LIN {X 0,Y 418.219,Z 282.716,A -85,B 0,C 180,E1 -10133.218,E2 -10133.218} C_VEL
LIN {X 0,Y 423.907,Z 299.688,A -85,B 0,C 180,E1 -10135.991,E2 -10135.991} C_VEL
LIN {X 0,Y 426.524,Z 308.051,A -85,B 0,C 180,E1 -10137.245,E2 -10137.245} C_VEL
LIN {X 0,Y 433.499,Z 322.682,A -85,B 0,C 180,E1 -10138.112,E2 -10138.112} C_VEL
LIN {X 0,Y 436.744,Z 342.587,A -85,B 0,C 180,E1 -10138.75,E2 -10138.75} C_VEL
LIN {X 0,Y 433.204,Z 515.05,A -85,B 0,C 180,E1 -10141.722,E2 -10141.722} C_VEL
LIN {X 0,Y 432.227,Z 531.382,A -85,B 0,C 180,E1 -10142.163,E2 -10142.163} C_VEL
LIN {X 0,Y 431.166,Z 547.235,A -85,B 0,C 180,E1 -10142.78,E2 -10142.78} C_VEL
LIN {X 0,Y 429.887,Z 562.43,A -85,B 0,C 180,E1 -10143.545,E2 -10143.545} C_VEL
LIN {X 0,Y 428.397,Z 577.584,A -85,B 0,C 180,E1 -10144.505,E2 -10144.505} C_VEL
LIN {X 0,Y 426.712,Z 592.691,A -85,B 0,C 180,E1 -10145.685,E2 -10145.685} C_VEL
LIN {X 0,Y 425.026,Z 606.696,A -85,B 0,C 180,E1 -10147.005,E2 -10147.005} C_VEL
LIN {X 0,Y 423.355,Z 620.63,A -85,B 0,C 180,E1 -10148.579,E2 -10148.579} C_VEL
LIN {X 0,Y 422.008,Z 631.644,A -85,B 0,C 180,E1 -10150.038,E2 -10150.038} C_VEL
LIN {X 0,Y 420.616,Z 642.771,A -85,B 0,C 180,E1 -10151.768,E2 -10151.768} C_VEL
LIN {X 0,Y 419.527,Z 653.245,A -85,B 0,C 180,E1 -10153.704,E2 -10153.704} C_VEL
LIN {X 0,Y 418.528,Z 662.163,A -85,B 0,C 180,E1 -10155.66,E2 -10155.66} C_VEL
LIN {X 0,Y 418.017,Z 668.813,A -85,B 0,C 180,E1 -10157.375,E2 -10157.375} C_VEL
LIN {X 0,Y 417.396,Z 676.506,A -85,B 0,C 180,E1 -10159.817,E2 -10159.817} C_VEL
LIN {X 0,Y 417.147,Z 682.365,A -85,B 0,C 180,E1 -10162.254,E2 -10162.254} C_VEL
LIN {X 0,Y 417.065,Z 685.793,A -85,B 0,C 180,E1 -10164.197,E2 -10164.197} C_VEL
LIN {X 0,Y 416.984,Z 688.283,A -85,B 0,C 180,E1 -10166.134,E2 -10166.134} C_VEL
LIN {X 0,Y 417.046,Z 689.691,A -85,B 0,C 180,E1 -10168.069,E2 -10168.069} C_VEL
LIN {X 0,Y 416.999,Z 690.219,A -85,B 0,C 180,E1 -10170,E2 -10170} C_VEL
LIN {X 0,Y 417.046,Z 689.689,A -85,B 0,C 180,E1 -10171.931,E2 -10171.931} C_VEL
LIN {X 0,Y 416.984,Z 688.278,A -85,B 0,C 180,E1 -10173.866,E2 -10173.866} C_VEL
LIN {X 0,Y 417.138,Z 685.094,A -85,B 0,C 180,E1 -10176.261,E2 -10176.261} C_VEL
LIN {X 0,Y 417.2,Z 681.284,A -85,B 0,C 180,E1 -10178.232,E2 -10178.232} C_VEL
LIN {X 0,Y 417.396,Z 676.5,A -85,B 0,C 180,E1 -10180.183,E2 -10180.183} C_VEL
LIN {X 0,Y 418.01,Z 668.8,A -85,B 0,C 180,E1 -10182.625,E2 -10182.625} C_VEL
LIN {X 0,Y 418.753,Z 660.111,A -85,B 0,C 180,E1 -10184.829,E2 -10184.829} C_VEL
LIN {X 0,Y 419.759,Z 650.785,A -85,B 0,C 180,E1 -10186.778,E2 -10186.778} C_VEL
LIN {X 0,Y 420.799,Z 641.099,A -85,B 0,C 180,E1 -10188.501,E2 -10188.501} C_VEL
LIN {X 0,Y 422.21,Z 629.874,A -85,B 0,C 180,E1 -10190.206,E2 -10190.206} C_VEL
LIN {X 0,Y 423.641,Z 618.18,A -85,B 0,C 180,E1 -10191.719,E2 -10191.719} C_VEL
LIN {X 0,Y 425.161,Z 605.467,A -85,B 0,C 180,E1 -10193.116,E2 -10193.116} C_VEL
LIN {X 0,Y 426.836,Z 591.192,A -85,B 0,C 180,E1 -10194.437,E2 -10194.437} C_VEL
LIN {X 0,Y 428.496,Z 576.432,A -85,B 0,C 180,E1 -10195.567,E2 -10195.567} C_VEL
LIN {X 0,Y 429.977,Z 561.328,A -85,B 0,C 180,E1 -10196.514,E2 -10196.514} C_VEL
LIN {X 0,Y 431.288,Z 545.808,A -85,B 0,C 180,E1 -10197.278,E2 -10197.278} C_VEL
LIN {X 0,Y 432.34,Z 530.29,A -85,B 0,C 180,E1 -10197.862,E2 -10197.862} C_VEL
LIN {X 0,Y 433.159,Z 515.027,A -85,B 0,C 180,E1 -10198.276,E2 -10198.276} C_VEL
LIN {X 0,Y 436.324,Z 361.208,A -85,B 0,C 180,E1 -10200.926,E2 -10200.926} C_VEL
LIN {X 0,Y 436.722,Z 342.306,A -85,B 0,C 180,E1 -10201.25,E2 -10201.25} C_VEL
LIN {X 0,Y 433.182,Z 322.055,A -85,B 0,C 180,E1 -10201.918,E2 -10201.918} C_VEL
LIN {X 0,Y 426.335,Z 307.543,A -85,B 0,C 180,E1 -10202.784,E2 -10202.784} C_VEL
LIN {X 0,Y 421.419,Z 292.204,A -85,B 0,C 180,E1 -10205.198,E2 -10205.198} C_VEL
LIN {X 0,Y 418.229,Z 282.702,A -85,B 0,C 180,E1 -10206.779,E2 -10206.779} C_VEL
LIN {X 0,Y 418.252,Z 282.699,A -85,B 0,C 180,E1 -10209.681,E2 -10209.681} C_VEL
LIN {X 0,Y 418.23,Z 282.699,A -85,B 0,C 180,E1 -10212.322,E2 -10212.322} C_VEL
LIN {X 0,Y 418.236,Z 282.699,A -85,B 0,C 180,E1 -10215.109,E2 -10215.109} C_VEL
LIN {X 0,Y 418.237,Z 282.694,A -85,B 0,C 180,E1 -10217.767,E2 -10217.767} C_VEL
LIN {X 0,Y 418.246,Z 282.692,A -85,B 0,C 180,E1 -10220.62,E2 -10220.62} C_VEL
LIN {X 0,Y 418.241,Z 282.695,A -85,B 0,C 180,E1 -10223.976,E2 -10223.976} C_VEL
LIN {X 0,Y 418.255,Z 282.695,A -85,B 0,C 180,E1 -10227.156,E2 -10227.156} C_VEL
LIN {X 0,Y 418.266,Z 282.695,A -85,B 0,C 180,E1 -10230.895,E2 -10230.895} C_VEL
LIN {X 0,Y 418.268,Z 282.694,A -85,B 0,C 180,E1 -10234.096,E2 -10234.096} C_VEL
LIN {X 0,Y 418.236,Z 282.701,A -85,B 0,C 180,E1 -10237.264,E2 -10237.264} C_VEL
LIN {X 0,Y 418.28,Z 282.673,A -85,B 0,C 180,E1 -10240.364,E2 -10240.364} C_VEL
LIN {X 0,Y 418.314,Z 282.69,A -85,B 0,C 180,E1 -10243.405,E2 -10243.405} C_VEL
LIN {X 0,Y 418.344,Z 282.666,A -85,B 0,C 180,E1 -10246.999,E2 -10246.999} C_VEL
LIN {X 0,Y 418.339,Z 282.685,A -85,B 0,C 180,E1 -10250.329,E2 -10250.329} C_VEL
LIN {X 0,Y 418.491,Z 282.646,A -85,B 0,C 180,E1 -10253.249,E2 -10253.249} C_VEL
LIN {X 0,Y 418.338,Z 282.676,A -85,B 0,C 180,E1 -10255.182,E2 -10255.182} C_VEL
LIN {X 0,Y 418.542,Z 282.658,A -85,B 0,C 180,E1 -10258.076,E2 -10258.076} C_VEL
LIN {X 0,Y 418.668,Z 282.628,A -85,B 0,C 180,E1 -10260,E2 -10260} C_VEL
LIN {X 0,Y 418.5,Z 282.659,A -85,B 0,C 180,E1 -10262.888,E2 -10262.888} C_VEL
LIN {X 0,Y 418.489,Z 282.655,A -85,B 0,C 180,E1 -10266.751,E2 -10266.751} C_VEL
LIN {X 0,Y 418.339,Z 282.679,A -85,B 0,C 180,E1 -10269.672,E2 -10269.672} C_VEL
LIN {X 0,Y 418.344,Z 282.682,A -85,B 0,C 180,E1 -10273.001,E2 -10273.001} C_VEL
LIN {X 0,Y 418.311,Z 282.678,A -85,B 0,C 180,E1 -10276.736,E2 -10276.736} C_VEL
LIN {X 0,Y 418.269,Z 282.69,A -85,B 0,C 180,E1 -10279.79,E2 -10279.79} C_VEL
LIN {X 0,Y 418.236,Z 282.682,A -85,B 0,C 180,E1 -10282.736,E2 -10282.736} C_VEL
LIN {X 0,Y 418.269,Z 282.692,A -85,B 0,C 180,E1 -10285.904,E2 -10285.904} C_VEL
LIN {X 0,Y 418.263,Z 282.689,A -85,B 0,C 180,E1 -10289.162,E2 -10289.162} C_VEL
LIN {X 0,Y 418.256,Z 282.698,A -85,B 0,C 180,E1 -10292.844,E2 -10292.844} C_VEL
LIN {X 0,Y 418.245,Z 282.697,A -85,B 0,C 180,E1 -10296.238,E2 -10296.238} C_VEL
LIN {X 0,Y 418.245,Z 282.695,A -85,B 0,C 180,E1 -10299.683,E2 -10299.683} C_VEL
LIN {X 0,Y 418.228,Z 282.688,A -85,B 0,C 180,E1 -10302.321,E2 -10302.321} C_VEL
LIN {X 0,Y 418.235,Z 282.693,A -85,B 0,C 180,E1 -10305.109,E2 -10305.109} C_VEL
LIN {X 0,Y 418.239,Z 282.699,A -85,B 0,C 180,E1 -10307.767,E2 -10307.767} C_VEL
LIN {X 0,Y 418.255,Z 282.701,A -85,B 0,C 180,E1 -10310.619,E2 -10310.619} C_VEL
LIN {X 0,Y 418.242,Z 282.685,A -85,B 0,C 180,E1 -10313.976,E2 -10313.976} C_VEL
LIN {X 0,Y 418.289,Z 282.829,A -85,B 0,C 180,E1 -10315.892,E2 -10315.892} C_VEL
LIN {X 0,Y 419.849,Z 287.641,A -85,B 0,C 180,E1 -10316.719,E2 -10316.719} C_VEL
LIN {X 0,Y 430.925,Z 308.814,A -85,B 0,C 180,E1 -10318.098,E2 -10318.098} C_VEL
LIN {X 0,Y 437.023,Z 321.625,A -85,B 0,C 180,E1 -10318.841,E2 -10318.841} C_VEL
LIN {X 0,Y 433.551,Z 490.007,A -85,B 0,C 180,E1 -10321.737,E2 -10321.737} C_VEL
LIN {X 0,Y 432.821,Z 506.702,A -85,B 0,C 180,E1 -10322.171,E2 -10322.171} C_VEL
LIN {X 0,Y 431.917,Z 522.513,A -85,B 0,C 180,E1 -10322.765,E2 -10322.765} C_VEL
LIN {X 0,Y 430.651,Z 538.1,A -85,B 0,C 180,E1 -10323.53,E2 -10323.53} C_VEL
LIN {X 0,Y 429.216,Z 553.749,A -85,B 0,C 180,E1 -10324.518,E2 -10324.518} C_VEL
LIN {X 0,Y 427.706,Z 567.977,A -85,B 0,C 180,E1 -10325.616,E2 -10325.616} C_VEL
LIN {X 0,Y 427.258,Z 572.266,A -85,B 0,C 180,E1 -10325.984,E2 -10325.984} C_VEL
LIN {X 0,Y 426.092,Z 577.23,A -85,B 0,C 180,E1 -10326.408,E2 -10326.408} C_VEL
LIN {X 0,Y 419.471,Z 591.273,A -85,B 0,C 180,E1 -10327.587,E2 -10327.587} C_VEL
LIN {X 0,Y 417.85,Z 595.77,A -85,B 0,C 180,E1 -10328.061,E2 -10328.061} C_VEL
LIN {X 0,Y 417.542,Z 597.202,A -85,B 0,C 180,E1 -10328.237,E2 -10328.237} C_VEL
LIN {X 0,Y 416.03,Z 608.35,A -85,B 0,C 180,E1 -10329.739,E2 -10329.739} C_VEL
LIN {X 0,Y 414.604,Z 619.332,A -85,B 0,C 180,E1 -10331.492,E2 -10331.492} C_VEL
LIN {X 0,Y 413.406,Z 628.464,A -85,B 0,C 180,E1 -10333.202,E2 -10333.202} C_VEL
LIN {X 0,Y 412.307,Z 637.483,A -85,B 0,C 180,E1 -10335.186,E2 -10335.186} C_VEL
LIN {X 0,Y 411.454,Z 645.015,A -85,B 0,C 180,E1 -10337.171,E2 -10337.171} C_VEL
LIN {X 0,Y 410.791,Z 651.178,A -85,B 0,C 180,E1 -10339.153,E2 -10339.153} C_VEL
LIN {X 0,Y 410.439,Z 656.225,A -85,B 0,C 180,E1 -10341.135,E2 -10341.135} C_VEL
LIN {X 0,Y 410.235,Z 660.129,A -85,B 0,C 180,E1 -10343.112,E2 -10343.112} C_VEL
LIN {X 0,Y 410.054,Z 663.037,A -85,B 0,C 180,E1 -10345.084,E2 -10345.084} C_VEL
LIN {X 0,Y 409.989,Z 664.945,A -85,B 0,C 180,E1 -10347.052,E2 -10347.052} C_VEL
LIN {X 0,Y 409.936,Z 665.915,A -85,B 0,C 180,E1 -10349.018,E2 -10349.018} C_VEL
LIN {X 0,Y 409.935,Z 665.931,A -85,B 0,C 180,E1 -10350.982,E2 -10350.982} C_VEL
LIN {X 0,Y 409.989,Z 665.022,A -85,B 0,C 180,E1 -10352.948,E2 -10352.948} C_VEL
LIN {X 0,Y 410.053,Z 663.144,A -85,B 0,C 180,E1 -10354.916,E2 -10354.916} C_VEL
LIN {X 0,Y 410.209,Z 660.297,A -85,B 0,C 180,E1 -10356.888,E2 -10356.888} C_VEL
LIN {X 0,Y 410.434,Z 656.422,A -85,B 0,C 180,E1 -10358.865,E2 -10358.865} C_VEL
LIN {X 0,Y 410.769,Z 651.443,A -85,B 0,C 180,E1 -10360.848,E2 -10360.848} C_VEL
LIN {X 0,Y 411.412,Z 645.349,A -85,B 0,C 180,E1 -10362.831,E2 -10362.831} C_VEL
LIN {X 0,Y 412.389,Z 636.862,A -85,B 0,C 180,E1 -10365.064,E2 -10365.064} C_VEL
LIN {X 0,Y 413.542,Z 627.7,A -85,B 0,C 180,E1 -10367.047,E2 -10367.047} C_VEL
LIN {X 0,Y 414.746,Z 618.27,A -85,B 0,C 180,E1 -10368.781,E2 -10368.781} C_VEL
LIN {X 0,Y 416.235,Z 607.27,A -85,B 0,C 180,E1 -10370.509,E2 -10370.509} C_VEL
LIN {X 0,Y 417.964,Z 594.32,A -85,B 0,C 180,E1 -10372.221,E2 -10372.221} C_VEL
LIN {X 0,Y 419.724,Z 580.937,A -85,B 0,C 180,E1 -10373.695,E2 -10373.695} C_VEL
LIN {X 0,Y 421.282,Z 567.819,A -85,B 0,C 180,E1 -10374.912,E2 -10374.912} C_VEL
LIN {X 0,Y 422.852,Z 553.19,A -85,B 0,C 180,E1 -10376.05,E2 -10376.05} C_VEL
LIN {X 0,Y 424.374,Z 537.721,A -85,B 0,C 180,E1 -10377.025,E2 -10377.025} C_VEL
LIN {X 0,Y 425.685,Z 522.027,A -85,B 0,C 180,E1 -10377.801,E2 -10377.801} C_VEL
LIN {X 0,Y 426.541,Z 506.841,A -85,B 0,C 180,E1 -10378.375,E2 -10378.375} C_VEL
LIN {X 0,Y 427.365,Z 489.44,A -85,B 0,C 180,E1 -10378.825,E2 -10378.825} C_VEL
LIN {X 0,Y 430.916,Z 323.696,A -85,B 0,C 180,E1 -10381.715,E2 -10381.715} C_VEL
LIN {X 0,Y 421.861,Z 305.105,A -85,B 0,C 180,E1 -10382.853,E2 -10382.853} C_VEL
LIN {X 0,Y 412.475,Z 287.59,A -85,B 0,C 180,E1 -10384.078,E2 -10384.078} C_VEL
LIN {X 0,Y 411.213,Z 283.577,A -85,B 0,C 180,E1 -10384.837,E2 -10384.837} C_VEL
LIN {X 0,Y 411.2,Z 283.576,A -85,B 0,C 180,E1 -10388.168,E2 -10388.168} C_VEL
LIN {X 0,Y 411.163,Z 283.584,A -85,B 0,C 180,E1 -10391.228,E2 -10391.228} C_VEL
LIN {X 0,Y 411.175,Z 283.58,A -85,B 0,C 180,E1 -10394.49,E2 -10394.49} C_VEL
LIN {X 0,Y 411.175,Z 283.575,A -85,B 0,C 180,E1 -10398.194,E2 -10398.194} C_VEL
LIN {X 0,Y 411.212,Z 283.574,A -85,B 0,C 180,E1 -10400.775,E2 -10400.775} C_VEL
LIN {X 0,Y 411.197,Z 283.574,A -85,B 0,C 180,E1 -10404.471,E2 -10404.471} C_VEL
LIN {X 0,Y 411.205,Z 283.567,A -85,B 0,C 180,E1 -10406.873,E2 -10406.873} C_VEL
LIN {X 0,Y 411.231,Z 283.573,A -85,B 0,C 180,E1 -10410.644,E2 -10410.644} C_VEL
LIN {X 0,Y 411.236,Z 283.567,A -85,B 0,C 180,E1 -10413.619,E2 -10413.619} C_VEL
LIN {X 0,Y 411.201,Z 283.566,A -85,B 0,C 180,E1 -10416.852,E2 -10416.852} C_VEL
LIN {X 0,Y 411.213,Z 283.572,A -85,B 0,C 180,E1 -10420.05,E2 -10420.05} C_VEL
LIN {X 0,Y 411.261,Z 283.553,A -85,B 0,C 180,E1 -10423.131,E2 -10423.131} C_VEL
LIN {X 0,Y 411.303,Z 283.564,A -85,B 0,C 180,E1 -10426.896,E2 -10426.896} C_VEL
LIN {X 0,Y 411.289,Z 283.545,A -85,B 0,C 180,E1 -10430.161,E2 -10430.161} C_VEL
LIN {X 0,Y 411.479,Z 283.533,A -85,B 0,C 180,E1 -10432.146,E2 -10432.146} C_VEL
LIN {X 0,Y 411.473,Z 283.54,A -85,B 0,C 180,E1 -10434.118,E2 -10434.118} C_VEL
LIN {X 0,Y 411.509,Z 283.522,A -85,B 0,C 180,E1 -10438.042,E2 -10438.042} C_VEL
LIN {X 0,Y 411.639,Z 283.519,A -85,B 0,C 180,E1 -10440,E2 -10440} C_VEL
LIN {X 0,Y 411.462,Z 283.527,A -85,B 0,C 180,E1 -10442.937,E2 -10442.937} C_VEL
LIN {X 0,Y 411.458,Z 283.545,A -85,B 0,C 180,E1 -10446.867,E2 -10446.867} C_VEL
LIN {X 0,Y 411.29,Z 283.549,A -85,B 0,C 180,E1 -10449.839,E2 -10449.839} C_VEL
LIN {X 0,Y 411.302,Z 283.565,A -85,B 0,C 180,E1 -10453.104,E2 -10453.104} C_VEL
LIN {X 0,Y 411.26,Z 283.573,A -85,B 0,C 180,E1 -10456.869,E2 -10456.869} C_VEL
LIN {X 0,Y 411.227,Z 283.572,A -85,B 0,C 180,E1 -10459.987,E2 -10459.987} C_VEL
LIN {X 0,Y 411.2,Z 283.579,A -85,B 0,C 180,E1 -10463.147,E2 -10463.147} C_VEL
LIN {X 0,Y 411.235,Z 283.575,A -85,B 0,C 180,E1 -10466.381,E2 -10466.381} C_VEL
LIN {X 0,Y 411.197,Z 283.576,A -85,B 0,C 180,E1 -10469.713,E2 -10469.713} C_VEL
LIN {X 0,Y 411.203,Z 283.579,A -85,B 0,C 180,E1 -10473.156,E2 -10473.156} C_VEL
LIN {X 0,Y 411.192,Z 283.581,A -85,B 0,C 180,E1 -10476.553,E2 -10476.553} C_VEL
LIN {X 0,Y 411.21,Z 283.578,A -85,B 0,C 180,E1 -10479.728,E2 -10479.728} C_VEL
LIN {X 0,Y 411.17,Z 283.584,A -85,B 0,C 180,E1 -10483.134,E2 -10483.134} C_VEL
LIN {X 0,Y 411.17,Z 283.582,A -85,B 0,C 180,E1 -10485.88,E2 -10485.88} C_VEL
LIN {X 0,Y 411.163,Z 283.584,A -85,B 0,C 180,E1 -10488.771,E2 -10488.771} C_VEL
LIN {X 0,Y 411.204,Z 283.577,A -85,B 0,C 180,E1 -10491.831,E2 -10491.831} C_VEL
LIN {X 0,Y 411.196,Z 283.652,A -85,B 0,C 180,E1 -10492.646,E2 -10492.646} C_VEL
LIN {X 0,Y 416.844,Z 300.376,A -85,B 0,C 180,E1 -10495.456,E2 -10495.456} C_VEL
LIN {X 0,Y 419.202,Z 307.76,A -85,B 0,C 180,E1 -10496.598,E2 -10496.598} C_VEL
LIN {X 0,Y 427.725,Z 325.536,A -85,B 0,C 180,E1 -10497.688,E2 -10497.688} C_VEL
LIN {X 0,Y 430.676,Z 343.856,A -85,B 0,C 180,E1 -10498.286,E2 -10498.286} C_VEL
LIN {X 0,Y 426.944,Z 515.303,A -85,B 0,C 180,E1 -10501.279,E2 -10501.279} C_VEL
LIN {X 0,Y 425.933,Z 531.184,A -85,B 0,C 180,E1 -10501.715,E2 -10501.715} C_VEL
LIN {X 0,Y 424.852,Z 547.035,A -85,B 0,C 180,E1 -10502.341,E2 -10502.341} C_VEL
LIN {X 0,Y 423.492,Z 562.227,A -85,B 0,C 180,E1 -10503.114,E2 -10503.114} C_VEL
LIN {X 0,Y 421.963,Z 577.256,A -85,B 0,C 180,E1 -10504.078,E2 -10504.078} C_VEL
LIN {X 0,Y 420.176,Z 592.485,A -85,B 0,C 180,E1 -10505.282,E2 -10505.282} C_VEL
LIN {X 0,Y 418.434,Z 606.49,A -85,B 0,C 180,E1 -10506.622,E2 -10506.622} C_VEL
LIN {X 0,Y 416.859,Z 618.789,A -85,B 0,C 180,E1 -10508.012,E2 -10508.012} C_VEL
LIN {X 0,Y 415.417,Z 629.701,A -85,B 0,C 180,E1 -10509.449,E2 -10509.449} C_VEL
LIN {X 0,Y 413.983,Z 640.917,A -85,B 0,C 180,E1 -10511.183,E2 -10511.183} C_VEL
LIN {X 0,Y 412.828,Z 650.742,A -85,B 0,C 180,E1 -10512.962,E2 -10512.962} C_VEL
LIN {X 0,Y 411.765,Z 659.918,A -85,B 0,C 180,E1 -10514.913,E2 -10514.913} C_VEL
LIN {X 0,Y 411.006,Z 668.604,A -85,B 0,C 180,E1 -10517.156,E2 -10517.156} C_VEL
LIN {X 0,Y 410.334,Z 676.298,A -85,B 0,C 180,E1 -10519.64,E2 -10519.64} C_VEL
LIN {X 0,Y 410.085,Z 682.158,A -85,B 0,C 180,E1 -10522.12,E2 -10522.12} C_VEL
LIN {X 0,Y 409.978,Z 685.585,A -85,B 0,C 180,E1 -10524.097,E2 -10524.097} C_VEL
LIN {X 0,Y 409.901,Z 688.076,A -85,B 0,C 180,E1 -10526.068,E2 -10526.068} C_VEL
LIN {X 0,Y 409.957,Z 689.484,A -85,B 0,C 180,E1 -10528.035,E2 -10528.035} C_VEL
LIN {X 0,Y 409.922,Z 690.012,A -85,B 0,C 180,E1 -10530,E2 -10530} C_VEL
LIN {X 0,Y 409.957,Z 689.481,A -85,B 0,C 180,E1 -10531.965,E2 -10531.965} C_VEL
LIN {X 0,Y 409.901,Z 688.071,A -85,B 0,C 180,E1 -10533.933,E2 -10533.933} C_VEL
LIN {X 0,Y 410.04,Z 685.1,A -85,B 0,C 180,E1 -10536.225,E2 -10536.225} C_VEL
LIN {X 0,Y 410.113,Z 681.074,A -85,B 0,C 180,E1 -10538.376,E2 -10538.376} C_VEL
LIN {X 0,Y 410.334,Z 676.29,A -85,B 0,C 180,E1 -10540.36,E2 -10540.36} C_VEL
LIN {X 0,Y 410.986,Z 668.589,A -85,B 0,C 180,E1 -10542.844,E2 -10542.844} C_VEL
LIN {X 0,Y 411.764,Z 659.899,A -85,B 0,C 180,E1 -10545.087,E2 -10545.087} C_VEL
LIN {X 0,Y 412.832,Z 650.711,A -85,B 0,C 180,E1 -10547.039,E2 -10547.039} C_VEL
LIN {X 0,Y 413.979,Z 640.887,A -85,B 0,C 180,E1 -10548.818,E2 -10548.818} C_VEL
LIN {X 0,Y 415.446,Z 629.661,A -85,B 0,C 180,E1 -10550.55,E2 -10550.55} C_VEL
LIN {X 0,Y 417.095,Z 616.775,A -85,B 0,C 180,E1 -10552.233,E2 -10552.233} C_VEL
LIN {X 0,Y 418.762,Z 604.076,A -85,B 0,C 180,E1 -10553.621,E2 -10553.621} C_VEL
LIN {X 0,Y 420.323,Z 590.979,A -85,B 0,C 180,E1 -10554.841,E2 -10554.841} C_VEL
LIN {X 0,Y 421.956,Z 577.191,A -85,B 0,C 180,E1 -10555.92,E2 -10555.92} C_VEL
LIN {X 0,Y 423.606,Z 561.114,A -85,B 0,C 180,E1 -10556.945,E2 -10556.945} C_VEL
LIN {X 0,Y 424.973,Z 545.593,A -85,B 0,C 180,E1 -10557.718,E2 -10557.718} C_VEL
LIN {X 0,Y 425.991,Z 530.99,A -85,B 0,C 180,E1 -10558.281,E2 -10558.281} C_VEL
LIN {X 0,Y 426.909,Z 515.208,A -85,B 0,C 180,E1 -10558.719,E2 -10558.719} C_VEL
LIN {X 0,Y 429.745,Z 385.05,A -85,B 0,C 180,E1 -10560.993,E2 -10560.993} C_VEL
LIN {X 0,Y 430.56,Z 343.103,A -85,B 0,C 180,E1 -10561.729,E2 -10561.729} C_VEL
LIN {X 0,Y 427.452,Z 325.048,A -85,B 0,C 180,E1 -10562.335,E2 -10562.335} C_VEL
LIN {X 0,Y 420.479,Z 310.409,A -85,B 0,C 180,E1 -10563.225,E2 -10563.225} C_VEL
LIN {X 0,Y 418.994,Z 307.145,A -85,B 0,C 180,E1 -10563.452,E2 -10563.452} C_VEL
LIN {X 0,Y 414.155,Z 292.202,A -85,B 0,C 180,E1 -10565.876,E2 -10565.876} C_VEL
LIN {X 0,Y 411.187,Z 283.58,A -85,B 0,C 180,E1 -10567.355,E2 -10567.355} C_VEL
LIN {X 0,Y 411.181,Z 283.58,A -85,B 0,C 180,E1 -10570.504,E2 -10570.504} C_VEL
LIN {X 0,Y 411.175,Z 283.579,A -85,B 0,C 180,E1 -10573.133,E2 -10573.133} C_VEL
LIN {X 0,Y 411.166,Z 283.576,A -85,B 0,C 180,E1 -10575.881,E2 -10575.881} C_VEL
LIN {X 0,Y 411.161,Z 283.576,A -85,B 0,C 180,E1 -10578.772,E2 -10578.772} C_VEL
LIN {X 0,Y 411.19,Z 283.571,A -85,B 0,C 180,E1 -10582.026,E2 -10582.026} C_VEL
LIN {X 0,Y 411.204,Z 283.574,A -85,B 0,C 180,E1 -10585.667,E2 -10585.667} C_VEL
LIN {X 0,Y 411.187,Z 283.578,A -85,B 0,C 180,E1 -10589.152,E2 -10589.152} C_VEL
LIN {X 0,Y 411.256,Z 283.567,A -85,B 0,C 180,E1 -10592.522,E2 -10592.522} C_VEL
LIN {X 0,Y 411.225,Z 283.571,A -85,B 0,C 180,E1 -10595.785,E2 -10595.785} C_VEL
LIN {X 0,Y 411.194,Z 283.563,A -85,B 0,C 180,E1 -10598.966,E2 -10598.966} C_VEL
LIN {X 0,Y 411.25,Z 283.566,A -85,B 0,C 180,E1 -10602.085,E2 -10602.085} C_VEL
LIN {X 0,Y 411.257,Z 283.556,A -85,B 0,C 180,E1 -10605.147,E2 -10605.147} C_VEL
LIN {X 0,Y 411.281,Z 283.557,A -85,B 0,C 180,E1 -10608.167,E2 -10608.167} C_VEL
LIN {X 0,Y 411.438,Z 283.536,A -85,B 0,C 180,E1 -10612.189,E2 -10612.189} C_VEL
LIN {X 0,Y 411.473,Z 283.521,A -85,B 0,C 180,E1 -10614.118,E2 -10614.118} C_VEL
LIN {X 0,Y 411.511,Z 283.534,A -85,B 0,C 180,E1 -10618.043,E2 -10618.043} C_VEL
LIN {X 0,Y 411.638,Z 283.503,A -85,B 0,C 180,E1 -10620,E2 -10620} C_VEL
LIN {X 0,Y 411.456,Z 283.536,A -85,B 0,C 180,E1 -10622.937,E2 -10622.937} C_VEL
LIN {X 0,Y 411.456,Z 283.528,A -85,B 0,C 180,E1 -10626.867,E2 -10626.867} C_VEL
LIN {X 0,Y 411.291,Z 283.557,A -85,B 0,C 180,E1 -10629.839,E2 -10629.839} C_VEL
LIN {X 0,Y 411.303,Z 283.557,A -85,B 0,C 180,E1 -10633.104,E2 -10633.104} C_VEL
LIN {X 0,Y 411.255,Z 283.559,A -85,B 0,C 180,E1 -10636.889,E2 -10636.889} C_VEL
LIN {X 0,Y 411.229,Z 283.567,A -85,B 0,C 180,E1 -10639.987,E2 -10639.987} C_VEL
LIN {X 0,Y 411.202,Z 283.565,A -85,B 0,C 180,E1 -10643.148,E2 -10643.148} C_VEL
LIN {X 0,Y 411.236,Z 283.568,A -85,B 0,C 180,E1 -10646.381,E2 -10646.381} C_VEL
LIN {X 0,Y 411.199,Z 283.574,A -85,B 0,C 180,E1 -10649.713,E2 -10649.713} C_VEL
LIN {X 0,Y 411.205,Z 283.576,A -85,B 0,C 180,E1 -10653.156,E2 -10653.156} C_VEL
LIN {X 0,Y 411.192,Z 283.575,A -85,B 0,C 180,E1 -10656.553,E2 -10656.553} C_VEL
LIN {X 0,Y 411.209,Z 283.571,A -85,B 0,C 180,E1 -10659.728,E2 -10659.728} C_VEL
LIN {X 0,Y 411.172,Z 283.573,A -85,B 0,C 180,E1 -10663.134,E2 -10663.134} C_VEL
LIN {X 0,Y 411.167,Z 283.569,A -85,B 0,C 180,E1 -10665.881,E2 -10665.881} C_VEL
LIN {X 0,Y 411.163,Z 283.583,A -85,B 0,C 180,E1 -10668.772,E2 -10668.772} C_VEL
LIN {X 0,Y 411.205,Z 283.559,A -85,B 0,C 180,E1 -10671.832,E2 -10671.832} C_VEL
LIN {X 0,Y 411.254,Z 283.734,A -85,B 0,C 180,E1 -10675.326,E2 -10675.326} C_VEL
LIN {X 0,Y 412.6,Z 287.923,A -85,B 0,C 180,E1 -10676.056,E2 -10676.056} C_VEL
LIN {X 0,Y 423.645,Z 308.558,A -85,B 0,C 180,E1 -10677.472,E2 -10677.472} C_VEL
LIN {X 0,Y 430.9,Z 323.77,A -85,B 0,C 180,E1 -10678.384,E2 -10678.384} C_VEL
LIN {X 0,Y 427.317,Z 490.405,A -85,B 0,C 180,E1 -10681.291,E2 -10681.291} C_VEL
LIN {X 0,Y 426.574,Z 506.922,A -85,B 0,C 180,E1 -10681.728,E2 -10681.728} C_VEL
LIN {X 0,Y 425.612,Z 522.73,A -85,B 0,C 180,E1 -10682.328,E2 -10682.328} C_VEL
LIN {X 0,Y 424.312,Z 538.316,A -85,B 0,C 180,E1 -10683.103,E2 -10683.103} C_VEL
LIN {X 0,Y 422.941,Z 552.775,A -85,B 0,C 180,E1 -10684.022,E2 -10684.022} C_VEL
LIN {X 0,Y 421.354,Z 566.772,A -85,B 0,C 180,E1 -10685.092,E2 -10685.092} C_VEL
LIN {X 0,Y 419.805,Z 580.075,A -85,B 0,C 180,E1 -10686.31,E2 -10686.31} C_VEL
LIN {X 0,Y 418.102,Z 593.096,A -85,B 0,C 180,E1 -10687.733,E2 -10687.733} C_VEL
LIN {X 0,Y 417.542,Z 597.202,A -85,B 0,C 180,E1 -10688.237,E2 -10688.237} C_VEL
LIN {X 0,Y 416.26,Z 601.604,A -85,B 0,C 180,E1 -10688.757,E2 -10688.757} C_VEL
LIN {X 0,Y 409.559,Z 614.004,A -85,B 0,C 180,E1 -10690.291,E2 -10690.291} C_VEL
LIN {X 0,Y 408.105,Z 617.806,A -85,B 0,C 180,E1 -10690.879,E2 -10690.879} C_VEL
LIN {X 0,Y 407.883,Z 619.044,A -85,B 0,C 180,E1 -10691.087,E2 -10691.087} C_VEL
LIN {X 0,Y 406.55,Z 628.675,A -85,B 0,C 180,E1 -10692.91,E2 -10692.91} C_VEL
LIN {X 0,Y 405.395,Z 637.694,A -85,B 0,C 180,E1 -10694.927,E2 -10694.927} C_VEL
LIN {X 0,Y 404.483,Z 645.226,A -85,B 0,C 180,E1 -10696.946,E2 -10696.946} C_VEL
LIN {X 0,Y 403.78,Z 651.388,A -85,B 0,C 180,E1 -10698.962,E2 -10698.962} C_VEL
LIN {X 0,Y 403.396,Z 656.435,A -85,B 0,C 180,E1 -10700.979,E2 -10700.979} C_VEL
LIN {X 0,Y 403.172,Z 660.337,A -85,B 0,C 180,E1 -10702.991,E2 -10702.991} C_VEL
LIN {X 0,Y 402.99,Z 663.244,A -85,B 0,C 180,E1 -10704.998,E2 -10704.998} C_VEL
LIN {X 0,Y 402.889,Z 665.153,A -85,B 0,C 180,E1 -10707,E2 -10707} C_VEL
LIN {X 0,Y 402.863,Z 666.122,A -85,B 0,C 180,E1 -10709,E2 -10709} C_VEL
LIN {X 0,Y 402.863,Z 666.137,A -85,B 0,C 180,E1 -10711,E2 -10711} C_VEL
LIN {X 0,Y 402.888,Z 665.229,A -85,B 0,C 180,E1 -10713,E2 -10713} C_VEL
LIN {X 0,Y 402.989,Z 663.35,A -85,B 0,C 180,E1 -10715.002,E2 -10715.002} C_VEL
LIN {X 0,Y 403.137,Z 660.504,A -85,B 0,C 180,E1 -10717.009,E2 -10717.009} C_VEL
LIN {X 0,Y 403.391,Z 656.629,A -85,B 0,C 180,E1 -10719.021,E2 -10719.021} C_VEL
LIN {X 0,Y 403.756,Z 651.65,A -85,B 0,C 180,E1 -10721.039,E2 -10721.039} C_VEL
LIN {X 0,Y 404.442,Z 645.556,A -85,B 0,C 180,E1 -10723.056,E2 -10723.056} C_VEL
LIN {X 0,Y 405.481,Z 637.069,A -85,B 0,C 180,E1 -10725.326,E2 -10725.326} C_VEL
LIN {X 0,Y 406.701,Z 627.907,A -85,B 0,C 180,E1 -10727.343,E2 -10727.343} C_VEL
LIN {X 0,Y 407.967,Z 618.477,A -85,B 0,C 180,E1 -10729.105,E2 -10729.105} C_VEL
LIN {X 0,Y 409.539,Z 607.476,A -85,B 0,C 180,E1 -10730.86,E2 -10730.86} C_VEL
LIN {X 0,Y 411.267,Z 595.116,A -85,B 0,C 180,E1 -10732.524,E2 -10732.524} C_VEL
LIN {X 0,Y 413.215,Z 581.14,A -85,B 0,C 180,E1 -10734.091,E2 -10734.091} C_VEL
LIN {X 0,Y 414.851,Z 568.021,A -85,B 0,C 180,E1 -10735.325,E2 -10735.325} C_VEL
LIN {X 0,Y 416.401,Z 554.059,A -85,B 0,C 180,E1 -10736.433,E2 -10736.433} C_VEL
LIN {X 0,Y 417.946,Z 539.027,A -85,B 0,C 180,E1 -10737.408,E2 -10737.408} C_VEL
LIN {X 0,Y 419.402,Z 522.225,A -85,B 0,C 180,E1 -10738.254,E2 -10738.254} C_VEL
LIN {X 0,Y 420.39,Z 506.12,A -85,B 0,C 180,E1 -10738.863,E2 -10738.863} C_VEL
LIN {X 0,Y 421.153,Z 490.021,A -85,B 0,C 180,E1 -10739.282,E2 -10739.282} C_VEL
LIN {X 0,Y 424.831,Z 325.708,A -85,B 0,C 180,E1 -10742.188,E2 -10742.188} C_VEL
LIN {X 0,Y 415.663,Z 307.15,A -85,B 0,C 180,E1 -10743.369,E2 -10743.369} C_VEL
LIN {X 0,Y 406.774,Z 290.718,A -85,B 0,C 180,E1 -10744.548,E2 -10744.548} C_VEL
LIN {X 0,Y 405.242,Z 287.751,A -85,B 0,C 180,E1 -10744.785,E2 -10744.785} C_VEL
LIN {X 0,Y 404.166,Z 284.441,A -85,B 0,C 180,E1 -10745.454,E2 -10745.454} C_VEL
LIN {X 0,Y 404.149,Z 284.457,A -85,B 0,C 180,E1 -10748.757,E2 -10748.757} C_VEL
LIN {X 0,Y 404.122,Z 284.456,A -85,B 0,C 180,E1 -10751.599,E2 -10751.599} C_VEL
LIN {X 0,Y 404.144,Z 284.456,A -85,B 0,C 180,E1 -10754.522,E2 -10754.522} C_VEL
LIN {X 0,Y 404.135,Z 284.459,A -85,B 0,C 180,E1 -10757.295,E2 -10757.295} C_VEL
LIN {X 0,Y 404.167,Z 284.45,A -85,B 0,C 180,E1 -10759.955,E2 -10759.955} C_VEL
LIN {X 0,Y 404.134,Z 284.447,A -85,B 0,C 180,E1 -10763.125,E2 -10763.125} C_VEL
LIN {X 0,Y 404.143,Z 284.451,A -85,B 0,C 180,E1 -10766.187,E2 -10766.187} C_VEL
LIN {X 0,Y 404.143,Z 284.455,A -85,B 0,C 180,E1 -10769.715,E2 -10769.715} C_VEL
LIN {X 0,Y 404.193,Z 284.437,A -85,B 0,C 180,E1 -10773.123,E2 -10773.123} C_VEL
LIN {X 0,Y 404.175,Z 284.452,A -85,B 0,C 180,E1 -10775.334,E2 -10775.334} C_VEL
LIN {X 0,Y 404.136,Z 284.439,A -85,B 0,C 180,E1 -10778.58,E2 -10778.58} C_VEL
LIN {X 0,Y 404.208,Z 284.443,A -85,B 0,C 180,E1 -10781.762,E2 -10781.762} C_VEL
LIN {X 0,Y 404.203,Z 284.43,A -85,B 0,C 180,E1 -10784.882,E2 -10784.882} C_VEL
LIN {X 0,Y 404.253,Z 284.438,A -85,B 0,C 180,E1 -10787.958,E2 -10787.958} C_VEL
LIN {X 0,Y 404.431,Z 284.411,A -85,B 0,C 180,E1 -10792.099,E2 -10792.099} C_VEL
LIN {X 0,Y 404.422,Z 284.419,A -85,B 0,C 180,E1 -10794.015,E2 -10794.015} C_VEL
LIN {X 0,Y 404.478,Z 284.398,A -85,B 0,C 180,E1 -10798.008,E2 -10798.008} C_VEL
LIN {X 0,Y 404.609,Z 284.395,A -85,B 0,C 180,E1 -10800,E2 -10800} C_VEL
LIN {X 0,Y 404.419,Z 284.403,A -85,B 0,C 180,E1 -10802.988,E2 -10802.988} C_VEL
LIN {X 0,Y 404.409,Z 284.425,A -85,B 0,C 180,E1 -10806.987,E2 -10806.987} C_VEL
LIN {X 0,Y 404.255,Z 284.424,A -85,B 0,C 180,E1 -10810.012,E2 -10810.012} C_VEL
LIN {X 0,Y 404.263,Z 284.443,A -85,B 0,C 180,E1 -10813.211,E2 -10813.211} C_VEL
LIN {X 0,Y 404.213,Z 284.449,A -85,B 0,C 180,E1 -10817.007,E2 -10817.007} C_VEL
LIN {X 0,Y 404.161,Z 284.454,A -85,B 0,C 180,E1 -10820.352,E2 -10820.352} C_VEL
LIN {X 0,Y 404.166,Z 284.452,A -85,B 0,C 180,E1 -10823.574,E2 -10823.574} C_VEL
LIN {X 0,Y 404.181,Z 284.452,A -85,B 0,C 180,E1 -10825.766,E2 -10825.766} C_VEL
LIN {X 0,Y 404.192,Z 284.449,A -85,B 0,C 180,E1 -10828,E2 -10828} C_VEL
LIN {X 0,Y 404.136,Z 284.46,A -85,B 0,C 180,E1 -10831.558,E2 -10831.558} C_VEL
LIN {X 0,Y 404.183,Z 284.453,A -85,B 0,C 180,E1 -10835.016,E2 -10835.016} C_VEL
LIN {X 0,Y 404.153,Z 284.46,A -85,B 0,C 180,E1 -10838.757,E2 -10838.757} C_VEL
LIN {X 0,Y 404.12,Z 284.462,A -85,B 0,C 180,E1 -10841.6,E2 -10841.6} C_VEL
LIN {X 0,Y 404.144,Z 284.461,A -85,B 0,C 180,E1 -10844.522,E2 -10844.522} C_VEL
LIN {X 0,Y 404.137,Z 284.46,A -85,B 0,C 180,E1 -10847.296,E2 -10847.296} C_VEL
LIN {X 0,Y 404.166,Z 284.454,A -85,B 0,C 180,E1 -10849.956,E2 -10849.956} C_VEL
LIN {X 0,Y 404.169,Z 284.527,A -85,B 0,C 180,E1 -10852.041,E2 -10852.041} C_VEL
LIN {X 0,Y 409.936,Z 301.312,A -85,B 0,C 180,E1 -10854.947,E2 -10854.947} C_VEL
LIN {X 0,Y 411.822,Z 307.346,A -85,B 0,C 180,E1 -10855.915,E2 -10855.915} C_VEL
LIN {X 0,Y 421.831,Z 328.016,A -85,B 0,C 180,E1 -10857.233,E2 -10857.233} C_VEL
LIN {X 0,Y 424.636,Z 344.718,A -85,B 0,C 180,E1 -10857.802,E2 -10857.802} C_VEL
LIN {X 0,Y 420.745,Z 514.575,A -85,B 0,C 180,E1 -10860.803,E2 -10860.803} C_VEL
LIN {X 0,Y 419.696,Z 530.986,A -85,B 0,C 180,E1 -10861.256,E2 -10861.256} C_VEL
LIN {X 0,Y 418.55,Z 546.833,A -85,B 0,C 180,E1 -10861.888,E2 -10861.888} C_VEL
LIN {X 0,Y 417.141,Z 562.024,A -85,B 0,C 180,E1 -10862.671,E2 -10862.671} C_VEL
LIN {X 0,Y 415.448,Z 577.956,A -85,B 0,C 180,E1 -10863.712,E2 -10863.712} C_VEL
LIN {X 0,Y 413.5,Z 593.711,A -85,B 0,C 180,E1 -10864.99,E2 -10864.99} C_VEL
LIN {X 0,Y 411.68,Z 607.462,A -85,B 0,C 180,E1 -10866.348,E2 -10866.348} C_VEL
LIN {X 0,Y 409.961,Z 620.214,A -85,B 0,C 180,E1 -10867.843,E2 -10867.843} C_VEL
LIN {X 0,Y 408.245,Z 632.865,A -85,B 0,C 180,E1 -10869.598,E2 -10869.598} C_VEL
LIN {X 0,Y 406.774,Z 643.653,A -85,B 0,C 180,E1 -10871.36,E2 -10871.36} C_VEL
LIN {X 0,Y 405.54,Z 654.068,A -85,B 0,C 180,E1 -10873.385,E2 -10873.385} C_VEL
LIN {X 0,Y 404.473,Z 662.762,A -85,B 0,C 180,E1 -10875.407,E2 -10875.407} C_VEL
LIN {X 0,Y 403.83,Z 670.129,A -85,B 0,C 180,E1 -10877.461,E2 -10877.461} C_VEL
LIN {X 0,Y 403.279,Z 676.089,A -85,B 0,C 180,E1 -10879.456,E2 -10879.456} C_VEL
LIN {X 0,Y 403.006,Z 681.95,A -85,B 0,C 180,E1 -10881.981,E2 -10881.981} C_VEL
LIN {X 0,Y 402.895,Z 685.378,A -85,B 0,C 180,E1 -10883.992,E2 -10883.992} C_VEL
LIN {X 0,Y 402.82,Z 687.869,A -85,B 0,C 180,E1 -10885.998,E2 -10885.998} C_VEL
LIN {X 0,Y 402.854,Z 689.276,A -85,B 0,C 180,E1 -10888.001,E2 -10888.001} C_VEL
LIN {X 0,Y 402.847,Z 689.805,A -85,B 0,C 180,E1 -10890,E2 -10890} C_VEL
LIN {X 0,Y 402.854,Z 689.274,A -85,B 0,C 180,E1 -10892,E2 -10892} C_VEL
LIN {X 0,Y 402.82,Z 687.863,A -85,B 0,C 180,E1 -10894.002,E2 -10894.002} C_VEL
LIN {X 0,Y 402.937,Z 685.116,A -85,B 0,C 180,E1 -10896.182,E2 -10896.182} C_VEL
LIN {X 0,Y 403.044,Z 680.864,A -85,B 0,C 180,E1 -10898.524,E2 -10898.524} C_VEL
LIN {X 0,Y 403.279,Z 676.08,A -85,B 0,C 180,E1 -10900.544,E2 -10900.544} C_VEL
LIN {X 0,Y 403.951,Z 668.377,A -85,B 0,C 180,E1 -10903.072,E2 -10903.072} C_VEL
LIN {X 0,Y 404.794,Z 659.687,A -85,B 0,C 180,E1 -10905.353,E2 -10905.353} C_VEL
LIN {X 0,Y 405.904,Z 650.551,A -85,B 0,C 180,E1 -10907.328,E2 -10907.328} C_VEL
LIN {X 0,Y 407.148,Z 640.674,A -85,B 0,C 180,E1 -10909.145,E2 -10909.145} C_VEL
LIN {X 0,Y 408.706,Z 629.448,A -85,B 0,C 180,E1 -10910.904,E2 -10910.904} C_VEL
LIN {X 0,Y 410.335,Z 617.319,A -85,B 0,C 180,E1 -10912.52,E2 -10912.52} C_VEL
LIN {X 0,Y 412.204,Z 603.864,A -85,B 0,C 180,E1 -10914.02,E2 -10914.02} C_VEL
LIN {X 0,Y 413.819,Z 590.766,A -85,B 0,C 180,E1 -10915.258,E2 -10915.258} C_VEL
LIN {X 0,Y 415.644,Z 576.014,A -85,B 0,C 180,E1 -10916.417,E2 -10916.417} C_VEL
LIN {X 0,Y 417.261,Z 560.9,A -85,B 0,C 180,E1 -10917.389,E2 -10917.389} C_VEL
LIN {X 0,Y 418.688,Z 545.379,A -85,B 0,C 180,E1 -10918.17,E2 -10918.17} C_VEL
LIN {X 0,Y 419.801,Z 529.854,A -85,B 0,C 180,E1 -10918.771,E2 -10918.771} C_VEL
LIN {X 0,Y 420.728,Z 514.394,A -85,B 0,C 180,E1 -10919.194,E2 -10919.194} C_VEL
LIN {X 0,Y 424.189,Z 360.278,A -85,B 0,C 180,E1 -10921.923,E2 -10921.923} C_VEL
LIN {X 0,Y 424.508,Z 343.959,A -85,B 0,C 180,E1 -10922.214,E2 -10922.214} C_VEL
LIN {X 0,Y 421.783,Z 327.963,A -85,B 0,C 180,E1 -10922.762,E2 -10922.762} C_VEL
LIN {X 0,Y 413.07,Z 309.88,A -85,B 0,C 180,E1 -10923.905,E2 -10923.905} C_VEL
LIN {X 0,Y 411.686,Z 306.997,A -85,B 0,C 180,E1 -10924.112,E2 -10924.112} C_VEL
LIN {X 0,Y 406.526,Z 291.515,A -85,B 0,C 180,E1 -10926.717,E2 -10926.717} C_VEL
LIN {X 0,Y 404.162,Z 284.453,A -85,B 0,C 180,E1 -10928.001,E2 -10928.001} C_VEL
LIN {X 0,Y 404.118,Z 284.459,A -85,B 0,C 180,E1 -10931.365,E2 -10931.365} C_VEL
LIN {X 0,Y 404.146,Z 284.451,A -85,B 0,C 180,E1 -10934.523,E2 -10934.523} C_VEL
LIN {X 0,Y 404.134,Z 284.456,A -85,B 0,C 180,E1 -10937.296,E2 -10937.296} C_VEL
LIN {X 0,Y 404.166,Z 284.446,A -85,B 0,C 180,E1 -10939.955,E2 -10939.955} C_VEL
LIN {X 0,Y 404.134,Z 284.452,A -85,B 0,C 180,E1 -10943.125,E2 -10943.125} C_VEL
LIN {X 0,Y 404.143,Z 284.452,A -85,B 0,C 180,E1 -10946.188,E2 -10946.188} C_VEL
LIN {X 0,Y 404.143,Z 284.451,A -85,B 0,C 180,E1 -10949.715,E2 -10949.715} C_VEL
LIN {X 0,Y 404.193,Z 284.448,A -85,B 0,C 180,E1 -10953.123,E2 -10953.123} C_VEL
LIN {X 0,Y 404.175,Z 284.45,A -85,B 0,C 180,E1 -10955.334,E2 -10955.334} C_VEL
LIN {X 0,Y 404.157,Z 284.446,A -85,B 0,C 180,E1 -10958.582,E2 -10958.582} C_VEL
LIN {X 0,Y 404.207,Z 284.444,A -85,B 0,C 180,E1 -10961.762,E2 -10961.762} C_VEL
LIN {X 0,Y 404.204,Z 284.438,A -85,B 0,C 180,E1 -10964.882,E2 -10964.882} C_VEL
LIN {X 0,Y 404.254,Z 284.432,A -85,B 0,C 180,E1 -10967.959,E2 -10967.959} C_VEL
LIN {X 0,Y 404.403,Z 284.412,A -85,B 0,C 180,E1 -10972.129,E2 -10972.129} C_VEL
LIN {X 0,Y 404.421,Z 284.398,A -85,B 0,C 180,E1 -10974.015,E2 -10974.015} C_VEL
LIN {X 0,Y 404.48,Z 284.41,A -85,B 0,C 180,E1 -10978.009,E2 -10978.009} C_VEL
LIN {X 0,Y 404.607,Z 284.378,A -85,B 0,C 180,E1 -10980,E2 -10980} C_VEL
LIN {X 0,Y 404.414,Z 284.414,A -85,B 0,C 180,E1 -10982.989,E2 -10982.989} C_VEL
LIN {X 0,Y 404.403,Z 284.404,A -85,B 0,C 180,E1 -10986.988,E2 -10986.988} C_VEL
LIN {X 0,Y 404.256,Z 284.433,A -85,B 0,C 180,E1 -10990.012,E2 -10990.012} C_VEL
LIN {X 0,Y 404.265,Z 284.433,A -85,B 0,C 180,E1 -10993.212,E2 -10993.212} C_VEL
LIN {X 0,Y 404.214,Z 284.437,A -85,B 0,C 180,E1 -10997.007,E2 -10997.007} C_VEL
LIN {X 0,Y 404.162,Z 284.446,A -85,B 0,C 180,E1 -11000.352,E2 -11000.352} C_VEL
LIN {X 0,Y 404.168,Z 284.449,A -85,B 0,C 180,E1 -11003.575,E2 -11003.575} C_VEL
LIN {X 0,Y 404.182,Z 284.447,A -85,B 0,C 180,E1 -11005.767,E2 -11005.767} C_VEL
LIN {X 0,Y 404.193,Z 284.428,A -85,B 0,C 180,E1 -11008,E2 -11008} C_VEL
LIN {X 0,Y 404.137,Z 284.451,A -85,B 0,C 180,E1 -11011.558,E2 -11011.558} C_VEL
LIN {X 0,Y 404.184,Z 284.449,A -85,B 0,C 180,E1 -11015.016,E2 -11015.016} C_VEL
LIN {X 0,Y 404.151,Z 284.44,A -85,B 0,C 180,E1 -11018.757,E2 -11018.757} C_VEL
LIN {X 0,Y 404.121,Z 284.447,A -85,B 0,C 180,E1 -11021.6,E2 -11021.6} C_VEL
LIN {X 0,Y 404.144,Z 284.457,A -85,B 0,C 180,E1 -11024.522,E2 -11024.522} C_VEL
LIN {X 0,Y 404.136,Z 284.459,A -85,B 0,C 180,E1 -11027.296,E2 -11027.296} C_VEL
LIN {X 0,Y 404.168,Z 284.452,A -85,B 0,C 180,E1 -11029.956,E2 -11029.956} C_VEL
LIN {X 0,Y 404.136,Z 284.431,A -85,B 0,C 180,E1 -11033.125,E2 -11033.125} C_VEL
LIN {X 0,Y 404.184,Z 284.596,A -85,B 0,C 180,E1 -11034.726,E2 -11034.726} C_VEL
LIN {X 0,Y 405.406,Z 288.172,A -85,B 0,C 180,E1 -11035.368,E2 -11035.368} C_VEL
LIN {X 0,Y 416.155,Z 308.152,A -85,B 0,C 180,E1 -11036.798,E2 -11036.798} C_VEL
LIN {X 0,Y 424.765,Z 325.782,A -85,B 0,C 180,E1 -11037.908,E2 -11037.908} C_VEL
LIN {X 0,Y 421.406,Z 480.521,A -85,B 0,C 180,E1 -11040.636,E2 -11040.636} C_VEL
LIN {X 0,Y 420.759,Z 498.999,A -85,B 0,C 180,E1 -11041.028,E2 -11041.028} C_VEL
LIN {X 0,Y 419.797,Z 515.62,A -85,B 0,C 180,E1 -11041.57,E2 -11041.57} C_VEL
LIN {X 0,Y 418.599,Z 531.786,A -85,B 0,C 180,E1 -11042.299,E2 -11042.299} C_VEL
LIN {X 0,Y 417.13,Z 547.359,A -85,B 0,C 180,E1 -11043.203,E2 -11043.203} C_VEL
LIN {X 0,Y 415.504,Z 562.564,A -85,B 0,C 180,E1 -11044.315,E2 -11044.315} C_VEL
LIN {X 0,Y 413.784,Z 576.47,A -85,B 0,C 180,E1 -11045.544,E2 -11045.544} C_VEL
LIN {X 0,Y 412.03,Z 589.423,A -85,B 0,C 180,E1 -11046.902,E2 -11046.902} C_VEL
LIN {X 0,Y 410.381,Z 601.501,A -85,B 0,C 180,E1 -11048.396,E2 -11048.396} C_VEL
LIN {X 0,Y 408.658,Z 613.407,A -85,B 0,C 180,E1 -11050.144,E2 -11050.144} C_VEL
LIN {X 0,Y 407.883,Z 619.044,A -85,B 0,C 180,E1 -11051.087,E2 -11051.087} C_VEL
LIN {X 0,Y 406.803,Z 622.77,A -85,B 0,C 180,E1 -11051.714,E2 -11051.714} C_VEL
LIN {X 0,Y 403.248,Z 628.709,A -85,B 0,C 180,E1 -11052.72,E2 -11052.72} C_VEL
LIN {X 0,Y 399.664,Z 634.213,A -85,B 0,C 180,E1 -11053.784,E2 -11053.784} C_VEL
LIN {X 0,Y 398.56,Z 637.259,A -85,B 0,C 180,E1 -11054.494,E2 -11054.494} C_VEL
LIN {X 0,Y 397.517,Z 645.436,A -85,B 0,C 180,E1 -11056.713,E2 -11056.713} C_VEL
LIN {X 0,Y 396.78,Z 651.598,A -85,B 0,C 180,E1 -11058.765,E2 -11058.765} C_VEL
LIN {X 0,Y 396.335,Z 656.644,A -85,B 0,C 180,E1 -11060.817,E2 -11060.817} C_VEL
LIN {X 0,Y 396.089,Z 660.546,A -85,B 0,C 180,E1 -11062.865,E2 -11062.865} C_VEL
LIN {X 0,Y 395.906,Z 663.452,A -85,B 0,C 180,E1 -11064.908,E2 -11064.908} C_VEL
LIN {X 0,Y 395.79,Z 665.361,A -85,B 0,C 180,E1 -11066.946,E2 -11066.946} C_VEL
LIN {X 0,Y 395.793,Z 666.329,A -85,B 0,C 180,E1 -11068.983,E2 -11068.983} C_VEL
LIN {X 0,Y 395.793,Z 666.344,A -85,B 0,C 180,E1 -11071.017,E2 -11071.017} C_VEL
LIN {X 0,Y 395.789,Z 665.436,A -85,B 0,C 180,E1 -11073.054,E2 -11073.054} C_VEL
LIN {X 0,Y 395.905,Z 663.558,A -85,B 0,C 180,E1 -11075.092,E2 -11075.092} C_VEL
LIN {X 0,Y 396.068,Z 660.711,A -85,B 0,C 180,E1 -11077.135,E2 -11077.135} C_VEL
LIN {X 0,Y 396.331,Z 656.837,A -85,B 0,C 180,E1 -11079.183,E2 -11079.183} C_VEL
LIN {X 0,Y 396.755,Z 651.857,A -85,B 0,C 180,E1 -11081.236,E2 -11081.236} C_VEL
LIN {X 0,Y 397.49,Z 645.763,A -85,B 0,C 180,E1 -11083.288,E2 -11083.288} C_VEL
LIN {X 0,Y 398.559,Z 637.276,A -85,B 0,C 180,E1 -11085.599,E2 -11085.599} C_VEL
LIN {X 0,Y 399.867,Z 628.114,A -85,B 0,C 180,E1 -11087.649,E2 -11087.649} C_VEL
LIN {X 0,Y 401.196,Z 618.683,A -85,B 0,C 180,E1 -11089.441,E2 -11089.441} C_VEL
LIN {X 0,Y 402.854,Z 607.681,A -85,B 0,C 180,E1 -11091.223,E2 -11091.223} C_VEL
LIN {X 0,Y 404.598,Z 595.848,A -85,B 0,C 180,E1 -11092.843,E2 -11092.843} C_VEL
LIN {X 0,Y 406.541,Z 582.511,A -85,B 0,C 180,E1 -11094.376,E2 -11094.376} C_VEL
LIN {X 0,Y 408.229,Z 569.644,A -85,B 0,C 180,E1 -11095.629,E2 -11095.629} C_VEL
LIN {X 0,Y 409.881,Z 555.712,A -85,B 0,C 180,E1 -11096.774,E2 -11096.774} C_VEL
LIN {X 0,Y 411.433,Z 541.222,A -85,B 0,C 180,E1 -11097.741,E2 -11097.741} C_VEL
LIN {X 0,Y 412.889,Z 526.313,A -85,B 0,C 180,E1 -11098.533,E2 -11098.533} C_VEL
LIN {X 0,Y 413.918,Z 510.884,A -85,B 0,C 180,E1 -11099.184,E2 -11099.184} C_VEL
LIN {X 0,Y 414.822,Z 494.862,A -85,B 0,C 180,E1 -11099.66,E2 -11099.66} C_VEL
LIN {X 0,Y 415.955,Z 449.134,A -85,B 0,C 180,E1 -11100.507,E2 -11100.507} C_VEL
LIN {X 0,Y 418.805,Z 327.873,A -85,B 0,C 180,E1 -11102.669,E2 -11102.669} C_VEL
LIN {X 0,Y 410.15,Z 310.418,A -85,B 0,C 180,E1 -11103.813,E2 -11103.813} C_VEL
LIN {X 0,Y 401.665,Z 294.692,A -85,B 0,C 180,E1 -11104.969,E2 -11104.969} C_VEL
LIN {X 0,Y 398.012,Z 287.943,A -85,B 0,C 180,E1 -11105.52,E2 -11105.52} C_VEL
LIN {X 0,Y 397.101,Z 285.313,A -85,B 0,C 180,E1 -11106.048,E2 -11106.048} C_VEL
LIN {X 0,Y 397.111,Z 285.327,A -85,B 0,C 180,E1 -11109.577,E2 -11109.577} C_VEL
LIN {X 0,Y 397.102,Z 285.332,A -85,B 0,C 180,E1 -11113.479,E2 -11113.479} C_VEL
LIN {X 0,Y 397.101,Z 285.329,A -85,B 0,C 180,E1 -11116.521,E2 -11116.521} C_VEL
LIN {X 0,Y 397.111,Z 285.329,A -85,B 0,C 180,E1 -11120.422,E2 -11120.422} C_VEL
LIN {X 0,Y 397.106,Z 285.329,A -85,B 0,C 180,E1 -11124.265,E2 -11124.265} C_VEL
LIN {X 0,Y 397.112,Z 285.322,A -85,B 0,C 180,E1 -11126.727,E2 -11126.727} C_VEL
LIN {X 0,Y 397.122,Z 285.329,A -85,B 0,C 180,E1 -11130.296,E2 -11130.296} C_VEL
LIN {X 0,Y 397.192,Z 285.304,A -85,B 0,C 180,E1 -11132.61,E2 -11132.61} C_VEL
LIN {X 0,Y 397.131,Z 285.325,A -85,B 0,C 180,E1 -11135.982,E2 -11135.982} C_VEL
LIN {X 0,Y 397.142,Z 285.326,A -85,B 0,C 180,E1 -11139.702,E2 -11139.702} C_VEL
LIN {X 0,Y 397.18,Z 285.31,A -85,B 0,C 180,E1 -11142.845,E2 -11142.845} C_VEL
LIN {X 0,Y 397.226,Z 285.316,A -85,B 0,C 180,E1 -11146.703,E2 -11146.703} C_VEL
LIN {X 0,Y 397.214,Z 285.299,A -85,B 0,C 180,E1 -11149.809,E2 -11149.809} C_VEL
LIN {X 0,Y 397.362,Z 285.297,A -85,B 0,C 180,E1 -11152.888,E2 -11152.888} C_VEL
LIN {X 0,Y 397.253,Z 285.311,A -85,B 0,C 180,E1 -11154.925,E2 -11154.925} C_VEL
LIN {X 0,Y 397.446,Z 285.272,A -85,B 0,C 180,E1 -11157.973,E2 -11157.973} C_VEL
LIN {X 0,Y 397.578,Z 285.271,A -85,B 0,C 180,E1 -11160,E2 -11160} C_VEL
LIN {X 0,Y 397.378,Z 285.279,A -85,B 0,C 180,E1 -11163.041,E2 -11163.041} C_VEL
LIN {X 0,Y 397.362,Z 285.303,A -85,B 0,C 180,E1 -11167.112,E2 -11167.112} C_VEL
LIN {X 0,Y 397.215,Z 285.299,A -85,B 0,C 180,E1 -11170.191,E2 -11170.191} C_VEL
LIN {X 0,Y 397.224,Z 285.318,A -85,B 0,C 180,E1 -11173.321,E2 -11173.321} C_VEL
LIN {X 0,Y 397.179,Z 285.323,A -85,B 0,C 180,E1 -11177.155,E2 -11177.155} C_VEL
LIN {X 0,Y 397.1,Z 285.334,A -85,B 0,C 180,E1 -11180.73,E2 -11180.73} C_VEL
LIN {X 0,Y 397.13,Z 285.328,A -85,B 0,C 180,E1 -11184.018,E2 -11184.018} C_VEL
LIN {X 0,Y 397.191,Z 285.321,A -85,B 0,C 180,E1 -11187.39,E2 -11187.39} C_VEL
LIN {X 0,Y 397.076,Z 285.339,A -85,B 0,C 180,E1 -11190.882,E2 -11190.882} C_VEL
LIN {X 0,Y 397.123,Z 285.336,A -85,B 0,C 180,E1 -11194.493,E2 -11194.493} C_VEL
LIN {X 0,Y 397.102,Z 285.338,A -85,B 0,C 180,E1 -11198.275,E2 -11198.275} C_VEL
LIN {X 0,Y 397.085,Z 285.341,A -85,B 0,C 180,E1 -11200.909,E2 -11200.909} C_VEL
LIN {X 0,Y 397.098,Z 285.336,A -85,B 0,C 180,E1 -11203.649,E2 -11203.649} C_VEL
LIN {X 0,Y 397.102,Z 285.337,A -85,B 0,C 180,E1 -11206.521,E2 -11206.521} C_VEL
LIN {X 0,Y 397.112,Z 285.335,A -85,B 0,C 180,E1 -11210.423,E2 -11210.423} C_VEL
LIN {X 0,Y 397.119,Z 285.362,A -85,B 0,C 180,E1 -11211.399,E2 -11211.399} C_VEL
LIN {X 0,Y 403.494,Z 303.906,A -85,B 0,C 180,E1 -11214.695,E2 -11214.695} C_VEL
LIN {X 0,Y 404.564,Z 307.284,A -85,B 0,C 180,E1 -11215.22,E2 -11215.22} C_VEL
LIN {X 0,Y 414.378,Z 327.056,A -85,B 0,C 180,E1 -11216.553,E2 -11216.553} C_VEL
LIN {X 0,Y 416.324,Z 331.446,A -85,B 0,C 180,E1 -11216.817,E2 -11216.817} C_VEL
LIN {X 0,Y 418.568,Z 345.436,A -85,B 0,C 180,E1 -11217.295,E2 -11217.295} C_VEL
LIN {X 0,Y 414.537,Z 514.764,A -85,B 0,C 180,E1 -11220.331,E2 -11220.331} C_VEL
LIN {X 0,Y 413.411,Z 531.706,A -85,B 0,C 180,E1 -11220.812,E2 -11220.812} C_VEL
LIN {X 0,Y 412.168,Z 547.936,A -85,B 0,C 180,E1 -11221.482,E2 -11221.482} C_VEL
LIN {X 0,Y 410.606,Z 563.813,A -85,B 0,C 180,E1 -11222.337,E2 -11222.337} C_VEL
LIN {X 0,Y 408.943,Z 578.626,A -85,B 0,C 180,E1 -11223.336,E2 -11223.336} C_VEL
LIN {X 0,Y 407.023,Z 593.506,A -85,B 0,C 180,E1 -11224.564,E2 -11224.564} C_VEL
LIN {X 0,Y 405.105,Z 607.256,A -85,B 0,C 180,E1 -11225.94,E2 -11225.94} C_VEL
LIN {X 0,Y 403.297,Z 620.006,A -85,B 0,C 180,E1 -11227.457,E2 -11227.457} C_VEL
LIN {X 0,Y 401.486,Z 632.657,A -85,B 0,C 180,E1 -11229.239,E2 -11229.239} C_VEL
LIN {X 0,Y 399.936,Z 643.444,A -85,B 0,C 180,E1 -11231.029,E2 -11231.029} C_VEL
LIN {X 0,Y 398.623,Z 653.859,A -85,B 0,C 180,E1 -11233.088,E2 -11233.088} C_VEL
LIN {X 0,Y 397.488,Z 662.553,A -85,B 0,C 180,E1 -11235.145,E2 -11235.145} C_VEL
LIN {X 0,Y 396.784,Z 670.14,A -85,B 0,C 180,E1 -11237.305,E2 -11237.305} C_VEL
LIN {X 0,Y 396.236,Z 675.881,A -85,B 0,C 180,E1 -11239.267,E2 -11239.267} C_VEL
LIN {X 0,Y 395.922,Z 681.741,A -85,B 0,C 180,E1 -11241.836,E2 -11241.836} C_VEL
LIN {X 0,Y 395.818,Z 685.17,A -85,B 0,C 180,E1 -11243.885,E2 -11243.885} C_VEL
LIN {X 0,Y 395.741,Z 687.662,A -85,B 0,C 180,E1 -11245.927,E2 -11245.927} C_VEL
LIN {X 0,Y 395.753,Z 689.069,A -85,B 0,C 180,E1 -11247.965,E2 -11247.965} C_VEL
LIN {X 0,Y 395.774,Z 689.599,A -85,B 0,C 180,E1 -11250,E2 -11250} C_VEL
LIN {X 0,Y 395.753,Z 689.066,A -85,B 0,C 180,E1 -11252.035,E2 -11252.035} C_VEL
LIN {X 0,Y 395.741,Z 687.656,A -85,B 0,C 180,E1 -11254.074,E2 -11254.074} C_VEL
LIN {X 0,Y 395.818,Z 685.163,A -85,B 0,C 180,E1 -11256.116,E2 -11256.116} C_VEL
LIN {X 0,Y 395.922,Z 681.734,A -85,B 0,C 180,E1 -11258.164,E2 -11258.164} C_VEL
LIN {X 0,Y 396.237,Z 675.869,A -85,B 0,C 180,E1 -11260.733,E2 -11260.733} C_VEL
LIN {X 0,Y 396.88,Z 668.816,A -85,B 0,C 180,E1 -11263.109,E2 -11263.109} C_VEL
LIN {X 0,Y 397.725,Z 660.494,A -85,B 0,C 180,E1 -11265.37,E2 -11265.37} C_VEL
LIN {X 0,Y 398.893,Z 651.344,A -85,B 0,C 180,E1 -11267.429,E2 -11267.429} C_VEL
LIN {X 0,Y 400.332,Z 640.461,A -85,B 0,C 180,E1 -11269.484,E2 -11269.484} C_VEL
LIN {X 0,Y 401.983,Z 629.235,A -85,B 0,C 180,E1 -11271.271,E2 -11271.271} C_VEL
LIN {X 0,Y 403.695,Z 617.005,A -85,B 0,C 180,E1 -11272.925,E2 -11272.925} C_VEL
LIN {X 0,Y 405.64,Z 603.65,A -85,B 0,C 180,E1 -11274.434,E2 -11274.434} C_VEL
LIN {X 0,Y 407.359,Z 590.637,A -85,B 0,C 180,E1 -11275.68,E2 -11275.68} C_VEL
LIN {X 0,Y 409.114,Z 577.038,A -85,B 0,C 180,E1 -11276.776,E2 -11276.776} C_VEL
LIN {X 0,Y 410.83,Z 561.687,A -85,B 0,C 180,E1 -11277.785,E2 -11277.785} C_VEL
LIN {X 0,Y 412.317,Z 546.466,A -85,B 0,C 180,E1 -11278.576,E2 -11278.576} C_VEL
LIN {X 0,Y 413.445,Z 531.471,A -85,B 0,C 180,E1 -11279.186,E2 -11279.186} C_VEL
LIN {X 0,Y 414.486,Z 515.43,A -85,B 0,C 180,E1 -11279.647,E2 -11279.647} C_VEL
LIN {X 0,Y 415.528,Z 469.85,A -85,B 0,C 180,E1 -11280.491,E2 -11280.491} C_VEL
LIN {X 0,Y 418.152,Z 360.928,A -85,B 0,C 180,E1 -11282.422,E2 -11282.422} C_VEL
LIN {X 0,Y 418.415,Z 344.637,A -85,B 0,C 180,E1 -11282.723,E2 -11282.723} C_VEL
LIN {X 0,Y 416.008,Z 330.654,A -85,B 0,C 180,E1 -11283.216,E2 -11283.216} C_VEL
LIN {X 0,Y 406.604,Z 311.184,A -85,B 0,C 180,E1 -11284.487,E2 -11284.487} C_VEL
LIN {X 0,Y 404.396,Z 306.841,A -85,B 0,C 180,E1 -11284.8,E2 -11284.8} C_VEL
LIN {X 0,Y 399.956,Z 293.751,A -85,B 0,C 180,E1 -11287.07,E2 -11287.07} C_VEL
LIN {X 0,Y 397.117,Z 285.334,A -85,B 0,C 180,E1 -11288.626,E2 -11288.626} C_VEL
LIN {X 0,Y 397.066,Z 285.337,A -85,B 0,C 180,E1 -11291.979,E2 -11291.979} C_VEL
LIN {X 0,Y 397.087,Z 285.333,A -85,B 0,C 180,E1 -11295.068,E2 -11295.068} C_VEL
LIN {X 0,Y 397.063,Z 285.33,A -85,B 0,C 180,E1 -11298.021,E2 -11298.021} C_VEL
LIN {X 0,Y 397.125,Z 285.326,A -85,B 0,C 180,E1 -11301.139,E2 -11301.139} C_VEL
LIN {X 0,Y 397.117,Z 285.326,A -85,B 0,C 180,E1 -11304.497,E2 -11304.497} C_VEL
LIN {X 0,Y 397.076,Z 285.333,A -85,B 0,C 180,E1 -11307.928,E2 -11307.928} C_VEL
LIN {X 0,Y 397.12,Z 285.331,A -85,B 0,C 180,E1 -11311.456,E2 -11311.456} C_VEL
LIN {X 0,Y 397.15,Z 285.326,A -85,B 0,C 180,E1 -11314.488,E2 -11314.488} C_VEL
LIN {X 0,Y 397.106,Z 285.327,A -85,B 0,C 180,E1 -11318.182,E2 -11318.182} C_VEL
LIN {X 0,Y 397.159,Z 285.315,A -85,B 0,C 180,E1 -11321.427,E2 -11321.427} C_VEL
LIN {X 0,Y 397.177,Z 285.318,A -85,B 0,C 180,E1 -11324.608,E2 -11324.608} C_VEL
LIN {X 0,Y 397.217,Z 285.305,A -85,B 0,C 180,E1 -11327.742,E2 -11327.742} C_VEL
LIN {X 0,Y 397.251,Z 285.314,A -85,B 0,C 180,E1 -11330.838,E2 -11330.838} C_VEL
LIN {X 0,Y 397.372,Z 285.274,A -85,B 0,C 180,E1 -11333.909,E2 -11333.909} C_VEL
LIN {X 0,Y 397.449,Z 285.286,A -85,B 0,C 180,E1 -11337.973,E2 -11337.973} C_VEL
LIN {X 0,Y 397.576,Z 285.253,A -85,B 0,C 180,E1 -11340,E2 -11340} C_VEL
LIN {X 0,Y 397.374,Z 285.291,A -85,B 0,C 180,E1 -11343.042,E2 -11343.042} C_VEL
LIN {X 0,Y 397.346,Z 285.286,A -85,B 0,C 180,E1 -11346.579,E2 -11346.579} C_VEL
LIN {X 0,Y 397.251,Z 285.293,A -85,B 0,C 180,E1 -11349.162,E2 -11349.162} C_VEL
LIN {X 0,Y 397.217,Z 285.317,A -85,B 0,C 180,E1 -11352.258,E2 -11352.258} C_VEL
LIN {X 0,Y 397.177,Z 285.3,A -85,B 0,C 180,E1 -11355.392,E2 -11355.392} C_VEL
LIN {X 0,Y 397.161,Z 285.325,A -85,B 0,C 180,E1 -11358.574,E2 -11358.574} C_VEL
LIN {X 0,Y 397.095,Z 285.309,A -85,B 0,C 180,E1 -11361.819,E2 -11361.819} C_VEL
LIN {X 0,Y 397.155,Z 285.327,A -85,B 0,C 180,E1 -11365.132,E2 -11365.132} C_VEL
LIN {X 0,Y 397.16,Z 285.303,A -85,B 0,C 180,E1 -11367.776,E2 -11367.776} C_VEL
LIN {X 0,Y 397.078,Z 285.338,A -85,B 0,C 180,E1 -11370.883,E2 -11370.883} C_VEL
LIN {X 0,Y 397.124,Z 285.327,A -85,B 0,C 180,E1 -11374.493,E2 -11374.493} C_VEL
LIN {X 0,Y 397.1,Z 285.315,A -85,B 0,C 180,E1 -11378.275,E2 -11378.275} C_VEL
LIN {X 0,Y 397.087,Z 285.329,A -85,B 0,C 180,E1 -11380.909,E2 -11380.909} C_VEL
LIN {X 0,Y 397.1,Z 285.331,A -85,B 0,C 180,E1 -11383.649,E2 -11383.649} C_VEL
LIN {X 0,Y 397.101,Z 285.324,A -85,B 0,C 180,E1 -11386.521,E2 -11386.521} C_VEL
LIN {X 0,Y 397.113,Z 285.333,A -85,B 0,C 180,E1 -11390.423,E2 -11390.423} C_VEL
LIN {X 0,Y 397.112,Z 285.35,A -85,B 0,C 180,E1 -11394.08,E2 -11394.08} C_VEL
LIN {X 0,Y 398.076,Z 288.233,A -85,B 0,C 180,E1 -11394.631,E2 -11394.631} C_VEL
LIN {X 0,Y 409.789,Z 309.69,A -85,B 0,C 180,E1 -11396.24,E2 -11396.24} C_VEL
LIN {X 0,Y 418.793,Z 328.105,A -85,B 0,C 180,E1 -11397.436,E2 -11397.436} C_VEL
LIN {X 0,Y 414.927,Z 491.405,A -85,B 0,C 180,E1 -11400.362,E2 -11400.362} C_VEL
LIN {X 0,Y 414.137,Z 507.363,A -85,B 0,C 180,E1 -11400.798,E2 -11400.798} C_VEL
LIN {X 0,Y 413.077,Z 523.164,A -85,B 0,C 180,E1 -11401.412,E2 -11401.412} C_VEL
LIN {X 0,Y 411.686,Z 538.747,A -85,B 0,C 180,E1 -11402.209,E2 -11402.209} C_VEL
LIN {X 0,Y 410.084,Z 554.218,A -85,B 0,C 180,E1 -11403.223,E2 -11403.223} C_VEL
LIN {X 0,Y 408.297,Z 568.618,A -85,B 0,C 180,E1 -11404.375,E2 -11404.375} C_VEL
LIN {X 0,Y 406.46,Z 582.833,A -85,B 0,C 180,E1 -11405.754,E2 -11405.754} C_VEL
LIN {X 0,Y 404.752,Z 594.688,A -85,B 0,C 180,E1 -11407.106,E2 -11407.106} C_VEL
LIN {X 0,Y 402.938,Z 607.034,A -85,B 0,C 180,E1 -11408.782,E2 -11408.782} C_VEL
LIN {X 0,Y 401.236,Z 618.145,A -85,B 0,C 180,E1 -11410.561,E2 -11410.561} C_VEL
LIN {X 0,Y 399.709,Z 628.887,A -85,B 0,C 180,E1 -11412.608,E2 -11412.608} C_VEL
LIN {X 0,Y 398.56,Z 637.259,A -85,B 0,C 180,E1 -11414.494,E2 -11414.494} C_VEL
LIN {X 0,Y 397.511,Z 640.225,A -85,B 0,C 180,E1 -11415.22,E2 -11415.22} C_VEL
LIN {X 0,Y 391.365,Z 648.256,A -85,B 0,C 180,E1 -11417.356,E2 -11417.356} C_VEL
LIN {X 0,Y 390.04,Z 650.636,A -85,B 0,C 180,E1 -11418.128,E2 -11418.128} C_VEL
LIN {X 0,Y 389.854,Z 651.359,A -85,B 0,C 180,E1 -11418.395,E2 -11418.395} C_VEL
LIN {X 0,Y 389.295,Z 656.854,A -85,B 0,C 180,E1 -11420.649,E2 -11420.649} C_VEL
LIN {X 0,Y 389.017,Z 660.755,A -85,B 0,C 180,E1 -11422.735,E2 -11422.735} C_VEL
LIN {X 0,Y 388.826,Z 663.66,A -85,B 0,C 180,E1 -11424.815,E2 -11424.815} C_VEL
LIN {X 0,Y 388.692,Z 665.569,A -85,B 0,C 180,E1 -11426.891,E2 -11426.891} C_VEL
LIN {X 0,Y 388.724,Z 666.535,A -85,B 0,C 180,E1 -11428.964,E2 -11428.964} C_VEL
LIN {X 0,Y 388.724,Z 666.55,A -85,B 0,C 180,E1 -11431.036,E2 -11431.036} C_VEL
LIN {X 0,Y 388.692,Z 665.643,A -85,B 0,C 180,E1 -11433.109,E2 -11433.109} C_VEL
LIN {X 0,Y 388.825,Z 663.765,A -85,B 0,C 180,E1 -11435.185,E2 -11435.185} C_VEL
LIN {X 0,Y 389.003,Z 660.918,A -85,B 0,C 180,E1 -11437.265,E2 -11437.265} C_VEL
LIN {X 0,Y 389.291,Z 657.044,A -85,B 0,C 180,E1 -11439.351,E2 -11439.351} C_VEL
LIN {X 0,Y 389.764,Z 652.064,A -85,B 0,C 180,E1 -11441.44,E2 -11441.44} C_VEL
LIN {X 0,Y 390.624,Z 645.391,A -85,B 0,C 180,E1 -11443.699,E2 -11443.699} C_VEL
LIN {X 0,Y 391.829,Z 636.418,A -85,B 0,C 180,E1 -11446.142,E2 -11446.142} C_VEL
LIN {X 0,Y 393.245,Z 627.1,A -85,B 0,C 180,E1 -11448.225,E2 -11448.225} C_VEL
LIN {X 0,Y 394.919,Z 615.943,A -85,B 0,C 180,E1 -11450.305,E2 -11450.305} C_VEL
LIN {X 0,Y 396.727,Z 604.348,A -85,B 0,C 180,E1 -11452.113,E2 -11452.113} C_VEL
LIN {X 0,Y 398.707,Z 591.65,A -85,B 0,C 180,E1 -11453.782,E2 -11453.782} C_VEL
LIN {X 0,Y 400.731,Z 577.817,A -85,B 0,C 180,E1 -11455.308,E2 -11455.308} C_VEL
LIN {X 0,Y 402.659,Z 564.118,A -85,B 0,C 180,E1 -11456.568,E2 -11456.568} C_VEL
LIN {X 0,Y 404.099,Z 551.158,A -85,B 0,C 180,E1 -11457.568,E2 -11457.568} C_VEL
LIN {X 0,Y 405.717,Z 536.068,A -85,B 0,C 180,E1 -11458.519,E2 -11458.519} C_VEL
LIN {X 0,Y 407.109,Z 520.485,A -85,B 0,C 180,E1 -11459.294,E2 -11459.294} C_VEL
LIN {X 0,Y 408.218,Z 503.749,A -85,B 0,C 180,E1 -11459.916,E2 -11459.916} C_VEL
LIN {X 0,Y 408.985,Z 486.842,A -85,B 0,C 180,E1 -11460.326,E2 -11460.326} C_VEL
LIN {X 0,Y 412.812,Z 330.255,A -85,B 0,C 180,E1 -11463.159,E2 -11463.159} C_VEL
LIN {X 0,Y 405.519,Z 315.336,A -85,B 0,C 180,E1 -11464.152,E2 -11464.152} C_VEL
LIN {X 0,Y 396.731,Z 298.943,A -85,B 0,C 180,E1 -11465.38,E2 -11465.38} C_VEL
LIN {X 0,Y 390.672,Z 288.284,A -85,B 0,C 180,E1 -11466.278,E2 -11466.278} C_VEL
LIN {X 0,Y 390.052,Z 286.189,A -85,B 0,C 180,E1 -11466.725,E2 -11466.725} C_VEL
LIN {X 0,Y 390.066,Z 286.207,A -85,B 0,C 180,E1 -11469.217,E2 -11469.217} C_VEL
LIN {X 0,Y 390.042,Z 286.205,A -85,B 0,C 180,E1 -11472.374,E2 -11472.374} C_VEL
LIN {X 0,Y 390.043,Z 286.204,A -85,B 0,C 180,E1 -11475.354,E2 -11475.354} C_VEL
LIN {X 0,Y 390.029,Z 286.21,A -85,B 0,C 180,E1 -11478.186,E2 -11478.186} C_VEL
LIN {X 0,Y 390.087,Z 286.207,A -85,B 0,C 180,E1 -11480.907,E2 -11480.907} C_VEL
LIN {X 0,Y 390.083,Z 286.206,A -85,B 0,C 180,E1 -11484.793,E2 -11484.793} C_VEL
LIN {X 0,Y 390.021,Z 286.207,A -85,B 0,C 180,E1 -11488.495,E2 -11488.495} C_VEL
LIN {X 0,Y 390.115,Z 286.186,A -85,B 0,C 180,E1 -11492.07,E2 -11492.07} C_VEL
LIN {X 0,Y 390.078,Z 286.206,A -85,B 0,C 180,E1 -11495.519,E2 -11495.519} C_VEL
LIN {X 0,Y 390.059,Z 286.194,A -85,B 0,C 180,E1 -11498.878,E2 -11498.878} C_VEL
LIN {X 0,Y 390.126,Z 286.197,A -85,B 0,C 180,E1 -11502.166,E2 -11502.166} C_VEL
LIN {X 0,Y 390.141,Z 286.189,A -85,B 0,C 180,E1 -11505.392,E2 -11505.392} C_VEL
LIN {X 0,Y 390.145,Z 286.195,A -85,B 0,C 180,E1 -11508.571,E2 -11508.571} C_VEL
LIN {X 0,Y 390.342,Z 286.166,A -85,B 0,C 180,E1 -11511.993,E2 -11511.993} C_VEL
LIN {X 0,Y 390.225,Z 286.187,A -85,B 0,C 180,E1 -11514.833,E2 -11514.833} C_VEL
LIN {X 0,Y 390.415,Z 286.147,A -85,B 0,C 180,E1 -11517.937,E2 -11517.937} C_VEL
LIN {X 0,Y 390.548,Z 286.147,A -85,B 0,C 180,E1 -11520,E2 -11520} C_VEL
LIN {X 0,Y 390.311,Z 286.157,A -85,B 0,C 180,E1 -11523.096,E2 -11523.096} C_VEL
LIN {X 0,Y 390.328,Z 286.171,A -85,B 0,C 180,E1 -11526.202,E2 -11526.202} C_VEL
LIN {X 0,Y 390.312,Z 286.177,A -85,B 0,C 180,E1 -11528.282,E2 -11528.282} C_VEL
LIN {X 0,Y 390.168,Z 286.189,A -85,B 0,C 180,E1 -11532.483,E2 -11532.483} C_VEL
LIN {X 0,Y 390.136,Z 286.197,A -85,B 0,C 180,E1 -11535.677,E2 -11535.677} C_VEL
LIN {X 0,Y 390.103,Z 286.204,A -85,B 0,C 180,E1 -11538.922,E2 -11538.922} C_VEL
LIN {X 0,Y 390.037,Z 286.211,A -85,B 0,C 180,E1 -11542.234,E2 -11542.234} C_VEL
LIN {X 0,Y 390.116,Z 286.205,A -85,B 0,C 180,E1 -11545.743,E2 -11545.743} C_VEL
LIN {X 0,Y 390.056,Z 286.214,A -85,B 0,C 180,E1 -11549.11,E2 -11549.11} C_VEL
LIN {X 0,Y 390.04,Z 286.215,A -85,B 0,C 180,E1 -11552.722,E2 -11552.722} C_VEL
LIN {X 0,Y 390.054,Z 286.21,A -85,B 0,C 180,E1 -11555.826,E2 -11555.826} C_VEL
LIN {X 0,Y 390.068,Z 286.215,A -85,B 0,C 180,E1 -11559.219,E2 -11559.219} C_VEL
LIN {X 0,Y 390.039,Z 286.218,A -85,B 0,C 180,E1 -11562.374,E2 -11562.374} C_VEL
LIN {X 0,Y 390.044,Z 286.215,A -85,B 0,C 180,E1 -11565.355,E2 -11565.355} C_VEL
LIN {X 0,Y 390.03,Z 286.216,A -85,B 0,C 180,E1 -11568.187,E2 -11568.187} C_VEL
LIN {X 0,Y 390.1,Z 286.272,A -85,B 0,C 180,E1 -11570.744,E2 -11570.744} C_VEL
LIN {X 0,Y 396.797,Z 305.764,A -85,B 0,C 180,E1 -11574.304,E2 -11574.304} C_VEL
LIN {X 0,Y 397.313,Z 307.118,A -85,B 0,C 180,E1 -11574.492,E2 -11574.492} C_VEL
LIN {X 0,Y 408.002,Z 328.47,A -85,B 0,C 180,E1 -11575.993,E2 -11575.993} C_VEL
LIN {X 0,Y 410.69,Z 334.623,A -85,B 0,C 180,E1 -11576.37,E2 -11576.37} C_VEL
LIN {X 0,Y 412.568,Z 347.525,A -85,B 0,C 180,E1 -11576.805,E2 -11576.805} C_VEL
LIN {X 0,Y 408.399,Z 514.078,A -85,B 0,C 180,E1 -11579.827,E2 -11579.827} C_VEL
LIN {X 0,Y 407.381,Z 529.675,A -85,B 0,C 180,E1 -11580.266,E2 -11580.266} C_VEL
LIN {X 0,Y 406.045,Z 546.432,A -85,B 0,C 180,E1 -11580.941,E2 -11580.941} C_VEL
LIN {X 0,Y 404.494,Z 561.617,A -85,B 0,C 180,E1 -11581.741,E2 -11581.741} C_VEL
LIN {X 0,Y 402.799,Z 576.601,A -85,B 0,C 180,E1 -11582.742,E2 -11582.742} C_VEL
LIN {X 0,Y 400.937,Z 590.614,A -85,B 0,C 180,E1 -11583.887,E2 -11583.887} C_VEL
LIN {X 0,Y 399.098,Z 603.512,A -85,B 0,C 180,E1 -11585.138,E2 -11585.138} C_VEL
LIN {X 0,Y 397.124,Z 616.855,A -85,B 0,C 180,E1 -11586.673,E2 -11586.673} C_VEL
LIN {X 0,Y 395.231,Z 629.076,A -85,B 0,C 180,E1 -11588.348,E2 -11588.348} C_VEL
LIN {X 0,Y 393.541,Z 640.29,A -85,B 0,C 180,E1 -11590.165,E2 -11590.165} C_VEL
LIN {X 0,Y 391.962,Z 651.163,A -85,B 0,C 180,E1 -11592.253,E2 -11592.253} C_VEL
LIN {X 0,Y 390.919,Z 659.29,A -85,B 0,C 180,E1 -11594.088,E2 -11594.088} C_VEL
LIN {X 0,Y 389.93,Z 667.976,A -85,B 0,C 180,E1 -11596.449,E2 -11596.449} C_VEL
LIN {X 0,Y 389.338,Z 674.239,A -85,B 0,C 180,E1 -11598.547,E2 -11598.547} C_VEL
LIN {X 0,Y 388.913,Z 679.372,A -85,B 0,C 180,E1 -11600.64,E2 -11600.64} C_VEL
LIN {X 0,Y 388.8,Z 683.368,A -85,B 0,C 180,E1 -11602.731,E2 -11602.731} C_VEL
LIN {X 0,Y 388.669,Z 686.324,A -85,B 0,C 180,E1 -11604.813,E2 -11604.813} C_VEL
LIN {X 0,Y 388.615,Z 688.27,A -85,B 0,C 180,E1 -11606.89,E2 -11606.89} C_VEL
LIN {X 0,Y 388.698,Z 689.238,A -85,B 0,C 180,E1 -11608.964,E2 -11608.964} C_VEL
LIN {X 0,Y 388.698,Z 689.237,A -85,B 0,C 180,E1 -11611.036,E2 -11611.036} C_VEL
LIN {X 0,Y 388.615,Z 688.265,A -85,B 0,C 180,E1 -11613.11,E2 -11613.11} C_VEL
LIN {X 0,Y 388.669,Z 686.316,A -85,B 0,C 180,E1 -11615.187,E2 -11615.187} C_VEL
LIN {X 0,Y 388.8,Z 683.359,A -85,B 0,C 180,E1 -11617.269,E2 -11617.269} C_VEL
LIN {X 0,Y 388.913,Z 679.364,A -85,B 0,C 180,E1 -11619.36,E2 -11619.36} C_VEL
LIN {X 0,Y 389.338,Z 674.224,A -85,B 0,C 180,E1 -11621.453,E2 -11621.453} C_VEL
LIN {X 0,Y 389.93,Z 667.954,A -85,B 0,C 180,E1 -11623.551,E2 -11623.551} C_VEL
LIN {X 0,Y 390.918,Z 659.263,A -85,B 0,C 180,E1 -11625.912,E2 -11625.912} C_VEL
LIN {X 0,Y 391.975,Z 651.13,A -85,B 0,C 180,E1 -11627.746,E2 -11627.746} C_VEL
LIN {X 0,Y 393.533,Z 640.248,A -85,B 0,C 180,E1 -11629.835,E2 -11629.835} C_VEL
LIN {X 0,Y 395.275,Z 629.023,A -85,B 0,C 180,E1 -11631.65,E2 -11631.65} C_VEL
LIN {X 0,Y 397.073,Z 616.792,A -85,B 0,C 180,E1 -11633.33,E2 -11633.33} C_VEL
LIN {X 0,Y 399.07,Z 603.436,A -85,B 0,C 180,E1 -11634.864,E2 -11634.864} C_VEL
LIN {X 0,Y 401.098,Z 589.29,A -85,B 0,C 180,E1 -11636.221,E2 -11636.221} C_VEL
LIN {X 0,Y 402.942,Z 575.228,A -85,B 0,C 180,E1 -11637.346,E2 -11637.346} C_VEL
LIN {X 0,Y 404.64,Z 560.472,A -85,B 0,C 180,E1 -11638.319,E2 -11638.319} C_VEL
LIN {X 0,Y 406.179,Z 544.948,A -85,B 0,C 180,E1 -11639.12,E2 -11639.12} C_VEL
LIN {X 0,Y 407.374,Z 529.418,A -85,B 0,C 180,E1 -11639.735,E2 -11639.735} C_VEL
LIN {X 0,Y 408.396,Z 512.997,A -85,B 0,C 180,E1 -11640.188,E2 -11640.188} C_VEL
LIN {X 0,Y 412.172,Z 360.229,A -85,B 0,C 180,E1 -11642.961,E2 -11642.961} C_VEL
LIN {X 0,Y 412.466,Z 346.014,A -85,B 0,C 180,E1 -11643.223,E2 -11643.223} C_VEL
LIN {X 0,Y 410.351,Z 333.636,A -85,B 0,C 180,E1 -11643.669,E2 -11643.669} C_VEL
LIN {X 0,Y 401.303,Z 314.828,A -85,B 0,C 180,E1 -11644.927,E2 -11644.927} C_VEL
LIN {X 0,Y 397.03,Z 306.522,A -85,B 0,C 180,E1 -11645.551,E2 -11645.551} C_VEL
LIN {X 0,Y 391.221,Z 289.767,A -85,B 0,C 180,E1 -11648.588,E2 -11648.588} C_VEL
LIN {X 0,Y 390.09,Z 286.206,A -85,B 0,C 180,E1 -11649.293,E2 -11649.293} C_VEL
LIN {X 0,Y 390.057,Z 286.21,A -85,B 0,C 180,E1 -11653.21,E2 -11653.21} C_VEL
LIN {X 0,Y 390.054,Z 286.206,A -85,B 0,C 180,E1 -11656.79,E2 -11656.79} C_VEL
LIN {X 0,Y 390.054,Z 286.206,A -85,B 0,C 180,E1 -11659.56,E2 -11659.56} C_VEL
LIN {X 0,Y 390.04,Z 286.206,A -85,B 0,C 180,E1 -11662.449,E2 -11662.449} C_VEL
LIN {X 0,Y 390.066,Z 286.206,A -85,B 0,C 180,E1 -11665.975,E2 -11665.975} C_VEL
LIN {X 0,Y 390.044,Z 286.206,A -85,B 0,C 180,E1 -11669.869,E2 -11669.869} C_VEL
LIN {X 0,Y 390.111,Z 286.202,A -85,B 0,C 180,E1 -11673.232,E2 -11673.232} C_VEL
LIN {X 0,Y 390.104,Z 286.204,A -85,B 0,C 180,E1 -11676.75,E2 -11676.75} C_VEL
LIN {X 0,Y 390.101,Z 286.18,A -85,B 0,C 180,E1 -11679.983,E2 -11679.983} C_VEL
LIN {X 0,Y 390.136,Z 286.202,A -85,B 0,C 180,E1 -11683.248,E2 -11683.248} C_VEL
LIN {X 0,Y 390.192,Z 286.168,A -85,B 0,C 180,E1 -11686.562,E2 -11686.562} C_VEL
LIN {X 0,Y 390.203,Z 286.193,A -85,B 0,C 180,E1 -11690.671,E2 -11690.671} C_VEL
LIN {X 0,Y 390.326,Z 286.15,A -85,B 0,C 180,E1 -11693.798,E2 -11693.798} C_VEL
LIN {X 0,Y 390.418,Z 286.162,A -85,B 0,C 180,E1 -11697.937,E2 -11697.937} C_VEL
LIN {X 0,Y 390.546,Z 286.128,A -85,B 0,C 180,E1 -11700,E2 -11700} C_VEL
LIN {X 0,Y 390.309,Z 286.172,A -85,B 0,C 180,E1 -11703.097,E2 -11703.097} C_VEL
LIN {X 0,Y 390.302,Z 286.165,A -85,B 0,C 180,E1 -11706.574,E2 -11706.574} C_VEL
LIN {X 0,Y 390.203,Z 286.172,A -85,B 0,C 180,E1 -11709.329,E2 -11709.329} C_VEL
LIN {X 0,Y 390.169,Z 286.196,A -85,B 0,C 180,E1 -11712.483,E2 -11712.483} C_VEL
LIN {X 0,Y 390.137,Z 286.177,A -85,B 0,C 180,E1 -11715.677,E2 -11715.677} C_VEL
LIN {X 0,Y 390.104,Z 286.206,A -85,B 0,C 180,E1 -11718.922,E2 -11718.922} C_VEL
LIN {X 0,Y 390.038,Z 286.188,A -85,B 0,C 180,E1 -11722.234,E2 -11722.234} C_VEL
LIN {X 0,Y 390.118,Z 286.199,A -85,B 0,C 180,E1 -11725.744,E2 -11725.744} C_VEL
LIN {X 0,Y 390.057,Z 286.199,A -85,B 0,C 180,E1 -11729.11,E2 -11729.11} C_VEL
LIN {X 0,Y 390.041,Z 286.21,A -85,B 0,C 180,E1 -11732.722,E2 -11732.722} C_VEL
LIN {X 0,Y 390.055,Z 286.207,A -85,B 0,C 180,E1 -11735.826,E2 -11735.826} C_VEL
LIN {X 0,Y 390.067,Z 286.2,A -85,B 0,C 180,E1 -11739.218,E2 -11739.218} C_VEL
LIN {X 0,Y 390.041,Z 286.198,A -85,B 0,C 180,E1 -11742.374,E2 -11742.374} C_VEL
LIN {X 0,Y 390.043,Z 286.202,A -85,B 0,C 180,E1 -11745.355,E2 -11745.355} C_VEL
LIN {X 0,Y 390.03,Z 286.214,A -85,B 0,C 180,E1 -11748.187,E2 -11748.187} C_VEL
LIN {X 0,Y 390.09,Z 286.204,A -85,B 0,C 180,E1 -11750.908,E2 -11750.908} C_VEL
LIN {X 0,Y 390.06,Z 286.284,A -85,B 0,C 180,E1 -11753.437,E2 -11753.437} C_VEL
LIN {X 0,Y 390.835,Z 288.651,A -85,B 0,C 180,E1 -11753.876,E2 -11753.876} C_VEL
LIN {X 0,Y 400.299,Z 305.444,A -85,B 0,C 180,E1 -11755.228,E2 -11755.228} C_VEL
LIN {X 0,Y 410.107,Z 324.547,A -85,B 0,C 180,E1 -11756.577,E2 -11756.577} C_VEL
LIN {X 0,Y 412.763,Z 330.219,A -85,B 0,C 180,E1 -11756.938,E2 -11756.938} C_VEL
LIN {X 0,Y 408.815,Z 490.657,A -85,B 0,C 180,E1 -11759.85,E2 -11759.85} C_VEL
LIN {X 0,Y 407.953,Z 507.583,A -85,B 0,C 180,E1 -11760.311,E2 -11760.311} C_VEL
LIN {X 0,Y 406.845,Z 523.381,A -85,B 0,C 180,E1 -11760.933,E2 -11760.933} C_VEL
LIN {X 0,Y 405.411,Z 538.963,A -85,B 0,C 180,E1 -11761.74,E2 -11761.74} C_VEL
LIN {X 0,Y 403.668,Z 555.13,A -85,B 0,C 180,E1 -11762.818,E2 -11762.818} C_VEL
LIN {X 0,Y 401.911,Z 568.831,A -85,B 0,C 180,E1 -11763.938,E2 -11763.938} C_VEL
LIN {X 0,Y 399.945,Z 583.046,A -85,B 0,C 180,E1 -11765.333,E2 -11765.333} C_VEL
LIN {X 0,Y 398.081,Z 595.494,A -85,B 0,C 180,E1 -11766.782,E2 -11766.782} C_VEL
LIN {X 0,Y 396.294,Z 607.245,A -85,B 0,C 180,E1 -11768.409,E2 -11768.409} C_VEL
LIN {X 0,Y 394.487,Z 618.357,A -85,B 0,C 180,E1 -11770.215,E2 -11770.215} C_VEL
LIN {X 0,Y 392.895,Z 629.098,A -85,B 0,C 180,E1 -11772.297,E2 -11772.297} C_VEL
LIN {X 0,Y 391.566,Z 638.116,A -85,B 0,C 180,E1 -11774.382,E2 -11774.382} C_VEL
LIN {X 0,Y 390.537,Z 645.648,A -85,B 0,C 180,E1 -11776.471,E2 -11776.471} C_VEL
LIN {X 0,Y 389.854,Z 651.359,A -85,B 0,C 180,E1 -11778.395,E2 -11778.395} C_VEL
LIN {X 0,Y 388.923,Z 653.561,A -85,B 0,C 180,E1 -11779.193,E2 -11779.193} C_VEL
LIN {X 0,Y 385.774,Z 656.832,A -85,B 0,C 180,E1 -11780.496,E2 -11780.496} C_VEL
LIN {X 0,Y 383.202,Z 659.156,A -85,B 0,C 180,E1 -11781.564,E2 -11781.564} C_VEL
LIN {X 0,Y 382.055,Z 660.659,A -85,B 0,C 180,E1 -11782.405,E2 -11782.405} C_VEL
LIN {X 0,Y 381.933,Z 661.103,A -85,B 0,C 180,E1 -11782.694,E2 -11782.694} C_VEL
LIN {X 0,Y 381.751,Z 663.868,A -85,B 0,C 180,E1 -11784.718,E2 -11784.718} C_VEL
LIN {X 0,Y 381.599,Z 665.776,A -85,B 0,C 180,E1 -11786.833,E2 -11786.833} C_VEL
LIN {X 0,Y 381.639,Z 666.742,A -85,B 0,C 180,E1 -11788.945,E2 -11788.945} C_VEL
LIN {X 0,Y 381.639,Z 666.757,A -85,B 0,C 180,E1 -11791.055,E2 -11791.055} C_VEL
LIN {X 0,Y 381.599,Z 665.85,A -85,B 0,C 180,E1 -11793.167,E2 -11793.167} C_VEL
LIN {X 0,Y 381.75,Z 663.972,A -85,B 0,C 180,E1 -11795.281,E2 -11795.281} C_VEL
LIN {X 0,Y 381.937,Z 661.125,A -85,B 0,C 180,E1 -11797.401,E2 -11797.401} C_VEL
LIN {X 0,Y 382.261,Z 657.251,A -85,B 0,C 180,E1 -11799.524,E2 -11799.524} C_VEL
LIN {X 0,Y 382.779,Z 652.271,A -85,B 0,C 180,E1 -11801.652,E2 -11801.652} C_VEL
LIN {X 0,Y 383.61,Z 646.001,A -85,B 0,C 180,E1 -11803.833,E2 -11803.833} C_VEL
LIN {X 0,Y 384.775,Z 637.691,A -85,B 0,C 180,E1 -11806.173,E2 -11806.173} C_VEL
LIN {X 0,Y 386.242,Z 628.589,A -85,B 0,C 180,E1 -11808.279,E2 -11808.279} C_VEL
LIN {X 0,Y 387.692,Z 619.097,A -85,B 0,C 180,E1 -11810.147,E2 -11810.147} C_VEL
LIN {X 0,Y 389.566,Z 608.092,A -85,B 0,C 180,E1 -11811.983,E2 -11811.983} C_VEL
LIN {X 0,Y 391.605,Z 595.505,A -85,B 0,C 180,E1 -11813.754,E2 -11813.754} C_VEL
LIN {X 0,Y 393.769,Z 581.753,A -85,B 0,C 180,E1 -11815.363,E2 -11815.363} C_VEL
LIN {X 0,Y 395.465,Z 570.049,A -85,B 0,C 180,E1 -11816.52,E2 -11816.52} C_VEL
LIN {X 0,Y 397.129,Z 556.805,A -85,B 0,C 180,E1 -11817.648,E2 -11817.648} C_VEL
LIN {X 0,Y 398.914,Z 541.623,A -85,B 0,C 180,E1 -11818.691,E2 -11818.691} C_VEL
LIN {X 0,Y 400.466,Z 526.709,A -85,B 0,C 180,E1 -11819.504,E2 -11819.504} C_VEL
LIN {X 0,Y 401.629,Z 510.359,A -85,B 0,C 180,E1 -11820.204,E2 -11820.204} C_VEL
LIN {X 0,Y 402.655,Z 493.958,A -85,B 0,C 180,E1 -11820.687,E2 -11820.687} C_VEL
LIN {X 0,Y 406.83,Z 333.283,A -85,B 0,C 180,E1 -11823.652,E2 -11823.652} C_VEL
LIN {X 0,Y 406.509,Z 331.707,A -85,B 0,C 180,E1 -11823.715,E2 -11823.715} C_VEL
LIN {X 0,Y 398.209,Z 315.001,A -85,B 0,C 180,E1 -11824.881,E2 -11824.881} C_VEL
LIN {X 0,Y 388.43,Z 297.13,A -85,B 0,C 180,E1 -11826.301,E2 -11826.301} C_VEL
LIN {X 0,Y 383.369,Z 288.521,A -85,B 0,C 180,E1 -11827.086,E2 -11827.086} C_VEL
LIN {X 0,Y 383,Z 287.071,A -85,B 0,C 180,E1 -11827.386,E2 -11827.386} C_VEL
LIN {X 0,Y 383.007,Z 287.083,A -85,B 0,C 180,E1 -11829.958,E2 -11829.958} C_VEL
LIN {X 0,Y 383.004,Z 287.081,A -85,B 0,C 180,E1 -11832.778,E2 -11832.778} C_VEL
LIN {X 0,Y 382.995,Z 287.082,A -85,B 0,C 180,E1 -11835.789,E2 -11835.789} C_VEL
LIN {X 0,Y 382.986,Z 287.082,A -85,B 0,C 180,E1 -11838.796,E2 -11838.796} C_VEL
LIN {X 0,Y 382.997,Z 287.084,A -85,B 0,C 180,E1 -11842.096,E2 -11842.096} C_VEL
LIN {X 0,Y 383.016,Z 287.088,A -85,B 0,C 180,E1 -11845.332,E2 -11845.332} C_VEL
LIN {X 0,Y 382.981,Z 287.089,A -85,B 0,C 180,E1 -11849.081,E2 -11849.081} C_VEL
LIN {X 0,Y 383.055,Z 287.065,A -85,B 0,C 180,E1 -11852.698,E2 -11852.698} C_VEL
LIN {X 0,Y 383.05,Z 287.085,A -85,B 0,C 180,E1 -11855.039,E2 -11855.039} C_VEL
LIN {X 0,Y 382.994,Z 287.071,A -85,B 0,C 180,E1 -11858.469,E2 -11858.469} C_VEL
LIN {X 0,Y 383.061,Z 287.077,A -85,B 0,C 180,E1 -11861.826,E2 -11861.826} C_VEL
LIN {X 0,Y 383.108,Z 287.059,A -85,B 0,C 180,E1 -11865.118,E2 -11865.118} C_VEL
LIN {X 0,Y 383.095,Z 287.075,A -85,B 0,C 180,E1 -11868.358,E2 -11868.358} C_VEL
LIN {X 0,Y 383.301,Z 287.043,A -85,B 0,C 180,E1 -11871.933,E2 -11871.933} C_VEL
LIN {X 0,Y 383.197,Z 287.064,A -85,B 0,C 180,E1 -11874.738,E2 -11874.738} C_VEL
LIN {X 0,Y 383.383,Z 287.022,A -85,B 0,C 180,E1 -11877.899,E2 -11877.899} C_VEL
LIN {X 0,Y 383.517,Z 287.022,A -85,B 0,C 180,E1 -11880,E2 -11880} C_VEL
LIN {X 0,Y 383.248,Z 287.036,A -85,B 0,C 180,E1 -11883.153,E2 -11883.153} C_VEL
LIN {X 0,Y 383.285,Z 287.049,A -85,B 0,C 180,E1 -11886.316,E2 -11886.316} C_VEL
LIN {X 0,Y 383.257,Z 287.056,A -85,B 0,C 180,E1 -11888.436,E2 -11888.436} C_VEL
LIN {X 0,Y 383.094,Z 287.064,A -85,B 0,C 180,E1 -11891.642,E2 -11891.642} C_VEL
LIN {X 0,Y 383.107,Z 287.074,A -85,B 0,C 180,E1 -11894.882,E2 -11894.882} C_VEL
LIN {X 0,Y 383.086,Z 287.075,A -85,B 0,C 180,E1 -11898.172,E2 -11898.172} C_VEL
LIN {X 0,Y 382.99,Z 287.088,A -85,B 0,C 180,E1 -11901.531,E2 -11901.531} C_VEL
LIN {X 0,Y 383.049,Z 287.084,A -85,B 0,C 180,E1 -11904.96,E2 -11904.96} C_VEL
LIN {X 0,Y 383.037,Z 287.088,A -85,B 0,C 180,E1 -11908.493,E2 -11908.493} C_VEL
LIN {X 0,Y 383.006,Z 287.093,A -85,B 0,C 180,E1 -11912.15,E2 -11912.15} C_VEL
LIN {X 0,Y 383.015,Z 287.094,A -85,B 0,C 180,E1 -11914.668,E2 -11914.668} C_VEL
LIN {X 0,Y 382.998,Z 287.093,A -85,B 0,C 180,E1 -11917.904,E2 -11917.904} C_VEL
LIN {X 0,Y 382.981,Z 287.097,A -85,B 0,C 180,E1 -11921.347,E2 -11921.347} C_VEL
LIN {X 0,Y 382.994,Z 287.095,A -85,B 0,C 180,E1 -11924.304,E2 -11924.304} C_VEL
LIN {X 0,Y 383.007,Z 287.093,A -85,B 0,C 180,E1 -11927.24,E2 -11927.24} C_VEL
LIN {X 0,Y 383.025,Z 287.126,A -85,B 0,C 180,E1 -11930.044,E2 -11930.044} C_VEL
LIN {X 0,Y 389.26,Z 305.005,A -85,B 0,C 180,E1 -11933.43,E2 -11933.43} C_VEL
LIN {X 0,Y 389.866,Z 306.696,A -85,B 0,C 180,E1 -11933.703,E2 -11933.703} C_VEL
LIN {X 0,Y 399.561,Z 325.551,A -85,B 0,C 180,E1 -11935.116,E2 -11935.116} C_VEL
LIN {X 0,Y 404.96,Z 337.178,A -85,B 0,C 180,E1 -11935.887,E2 -11935.887} C_VEL
LIN {X 0,Y 406.619,Z 348.272,A -85,B 0,C 180,E1 -11936.274,E2 -11936.274} C_VEL
LIN {X 0,Y 402.269,Z 514.357,A -85,B 0,C 180,E1 -11939.33,E2 -11939.33} C_VEL
LIN {X 0,Y 401.151,Z 530.395,A -85,B 0,C 180,E1 -11939.792,E2 -11939.792} C_VEL
LIN {X 0,Y 399.847,Z 546.232,A -85,B 0,C 180,E1 -11940.446,E2 -11940.446} C_VEL
LIN {X 0,Y 398.251,Z 561.415,A -85,B 0,C 180,E1 -11941.257,E2 -11941.257} C_VEL
LIN {X 0,Y 396.465,Z 576.39,A -85,B 0,C 180,E1 -11942.269,E2 -11942.269} C_VEL
LIN {X 0,Y 394.514,Z 590.507,A -85,B 0,C 180,E1 -11943.439,E2 -11943.439} C_VEL
LIN {X 0,Y 392.546,Z 603.304,A -85,B 0,C 180,E1 -11944.694,E2 -11944.694} C_VEL
LIN {X 0,Y 390.517,Z 616.648,A -85,B 0,C 180,E1 -11946.255,E2 -11946.255} C_VEL
LIN {X 0,Y 388.572,Z 628.869,A -85,B 0,C 180,E1 -11947.957,E2 -11947.957} C_VEL
LIN {X 0,Y 386.772,Z 640.082,A -85,B 0,C 180,E1 -11949.803,E2 -11949.803} C_VEL
LIN {X 0,Y 385.081,Z 650.953,A -85,B 0,C 180,E1 -11951.925,E2 -11951.925} C_VEL
LIN {X 0,Y 384.005,Z 659.081,A -85,B 0,C 180,E1 -11953.793,E2 -11953.793} C_VEL
LIN {X 0,Y 382.937,Z 667.767,A -85,B 0,C 180,E1 -11956.197,E2 -11956.197} C_VEL
LIN {X 0,Y 382.296,Z 674.03,A -85,B 0,C 180,E1 -11958.333,E2 -11958.333} C_VEL
LIN {X 0,Y 381.857,Z 679.164,A -85,B 0,C 180,E1 -11960.466,E2 -11960.466} C_VEL
LIN {X 0,Y 381.7,Z 683.16,A -85,B 0,C 180,E1 -11962.595,E2 -11962.595} C_VEL
LIN {X 0,Y 381.579,Z 686.117,A -85,B 0,C 180,E1 -11964.716,E2 -11964.716} C_VEL
LIN {X 0,Y 381.526,Z 688.063,A -85,B 0,C 180,E1 -11966.832,E2 -11966.832} C_VEL
LIN {X 0,Y 381.612,Z 689.031,A -85,B 0,C 180,E1 -11968.945,E2 -11968.945} C_VEL
LIN {X 0,Y 381.612,Z 689.03,A -85,B 0,C 180,E1 -11971.055,E2 -11971.055} C_VEL
LIN {X 0,Y 381.527,Z 688.057,A -85,B 0,C 180,E1 -11973.168,E2 -11973.168} C_VEL
LIN {X 0,Y 381.579,Z 686.108,A -85,B 0,C 180,E1 -11975.284,E2 -11975.284} C_VEL
LIN {X 0,Y 381.7,Z 683.15,A -85,B 0,C 180,E1 -11977.405,E2 -11977.405} C_VEL
LIN {X 0,Y 381.857,Z 679.154,A -85,B 0,C 180,E1 -11979.535,E2 -11979.535} C_VEL
LIN {X 0,Y 382.296,Z 674.013,A -85,B 0,C 180,E1 -11981.667,E2 -11981.667} C_VEL
LIN {X 0,Y 382.936,Z 667.743,A -85,B 0,C 180,E1 -11983.803,E2 -11983.803} C_VEL
LIN {X 0,Y 384.003,Z 659.052,A -85,B 0,C 180,E1 -11986.207,E2 -11986.207} C_VEL
LIN {X 0,Y 385.337,Z 649.612,A -85,B 0,C 180,E1 -11988.352,E2 -11988.352} C_VEL
LIN {X 0,Y 386.759,Z 640.036,A -85,B 0,C 180,E1 -11990.197,E2 -11990.197} C_VEL
LIN {X 0,Y 388.614,Z 628.811,A -85,B 0,C 180,E1 -11992.04,E2 -11992.04} C_VEL
LIN {X 0,Y 390.501,Z 616.58,A -85,B 0,C 180,E1 -11993.746,E2 -11993.746} C_VEL
LIN {X 0,Y 392.556,Z 603.223,A -85,B 0,C 180,E1 -11995.305,E2 -11995.305} C_VEL
LIN {X 0,Y 394.653,Z 589.32,A -85,B 0,C 180,E1 -11996.659,E2 -11996.659} C_VEL
LIN {X 0,Y 396.463,Z 576.254,A -85,B 0,C 180,E1 -11997.731,E2 -11997.731} C_VEL
LIN {X 0,Y 398.256,Z 561.259,A -85,B 0,C 180,E1 -11998.743,E2 -11998.743} C_VEL
LIN {X 0,Y 399.849,Z 546.036,A -85,B 0,C 180,E1 -11999.554,E2 -11999.554} C_VEL
LIN {X 0,Y 401.147,Z 530.118,A -85,B 0,C 180,E1 -12000.208,E2 -12000.208} C_VEL
LIN {X 0,Y 402.227,Z 514.103,A -85,B 0,C 180,E1 -12000.669,E2 -12000.669} C_VEL
LIN {X 0,Y 406.211,Z 360.56,A -85,B 0,C 180,E1 -12003.496,E2 -12003.496} C_VEL
LIN {X 0,Y 406.552,Z 347.16,A -85,B 0,C 180,E1 -12003.743,E2 -12003.743} C_VEL
LIN {X 0,Y 404.665,Z 336.416,A -85,B 0,C 180,E1 -12004.145,E2 -12004.145} C_VEL
LIN {X 0,Y 395.864,Z 318.184,A -85,B 0,C 180,E1 -12005.401,E2 -12005.401} C_VEL
LIN {X 0,Y 389.675,Z 306.285,A -85,B 0,C 180,E1 -12006.323,E2 -12006.323} C_VEL
LIN {X 0,Y 383.893,Z 289.633,A -85,B 0,C 180,E1 -12009.446,E2 -12009.446} C_VEL
LIN {X 0,Y 383.027,Z 287.088,A -85,B 0,C 180,E1 -12009.956,E2 -12009.956} C_VEL
LIN {X 0,Y 383.003,Z 287.086,A -85,B 0,C 180,E1 -12012.779,E2 -12012.779} C_VEL
LIN {X 0,Y 382.995,Z 287.085,A -85,B 0,C 180,E1 -12015.789,E2 -12015.789} C_VEL
LIN {X 0,Y 382.985,Z 287.085,A -85,B 0,C 180,E1 -12018.796,E2 -12018.796} C_VEL
LIN {X 0,Y 382.996,Z 287.083,A -85,B 0,C 180,E1 -12022.096,E2 -12022.096} C_VEL
LIN {X 0,Y 383.015,Z 287.083,A -85,B 0,C 180,E1 -12025.332,E2 -12025.332} C_VEL
LIN {X 0,Y 382.98,Z 287.092,A -85,B 0,C 180,E1 -12029.081,E2 -12029.081} C_VEL
LIN {X 0,Y 383.054,Z 287.079,A -85,B 0,C 180,E1 -12032.698,E2 -12032.698} C_VEL
LIN {X 0,Y 383.05,Z 287.082,A -85,B 0,C 180,E1 -12035.04,E2 -12035.04} C_VEL
LIN {X 0,Y 382.997,Z 287.082,A -85,B 0,C 180,E1 -12038.469,E2 -12038.469} C_VEL
LIN {X 0,Y 383.087,Z 287.075,A -85,B 0,C 180,E1 -12041.828,E2 -12041.828} C_VEL
LIN {X 0,Y 383.108,Z 287.06,A -85,B 0,C 180,E1 -12045.118,E2 -12045.118} C_VEL
LIN {X 0,Y 383.095,Z 287.068,A -85,B 0,C 180,E1 -12048.358,E2 -12048.358} C_VEL
LIN {X 0,Y 383.262,Z 287.045,A -85,B 0,C 180,E1 -12051.976,E2 -12051.976} C_VEL
LIN {X 0,Y 383.197,Z 287.045,A -85,B 0,C 180,E1 -12054.739,E2 -12054.739} C_VEL
LIN {X 0,Y 383.386,Z 287.038,A -85,B 0,C 180,E1 -12057.899,E2 -12057.899} C_VEL
LIN {X 0,Y 383.515,Z 287.002,A -85,B 0,C 180,E1 -12060,E2 -12060} C_VEL
LIN {X 0,Y 383.245,Z 287.052,A -85,B 0,C 180,E1 -12063.154,E2 -12063.154} C_VEL
LIN {X 0,Y 383.263,Z 287.042,A -85,B 0,C 180,E1 -12066.565,E2 -12066.565} C_VEL
LIN {X 0,Y 383.15,Z 287.053,A -85,B 0,C 180,E1 -12069.502,E2 -12069.502} C_VEL
LIN {X 0,Y 383.123,Z 287.062,A -85,B 0,C 180,E1 -12073.536,E2 -12073.536} C_VEL
LIN {X 0,Y 383.093,Z 287.075,A -85,B 0,C 180,E1 -12077.455,E2 -12077.455} C_VEL
LIN {X 0,Y 383.027,Z 287.07,A -85,B 0,C 180,E1 -12080.647,E2 -12080.647} C_VEL
LIN {X 0,Y 383.032,Z 287.081,A -85,B 0,C 180,E1 -12083.808,E2 -12083.808} C_VEL
LIN {X 0,Y 383.078,Z 287.076,A -85,B 0,C 180,E1 -12086.124,E2 -12086.124} C_VEL
LIN {X 0,Y 382.991,Z 287.088,A -85,B 0,C 180,E1 -12089.7,E2 -12089.7} C_VEL
LIN {X 0,Y 383.002,Z 287.088,A -85,B 0,C 180,E1 -12093.401,E2 -12093.401} C_VEL
LIN {X 0,Y 383.031,Z 287.083,A -85,B 0,C 180,E1 -12096.165,E2 -12096.165} C_VEL
LIN {X 0,Y 383.007,Z 287.085,A -85,B 0,C 180,E1 -12099.959,E2 -12099.959} C_VEL
LIN {X 0,Y 383.004,Z 287.076,A -85,B 0,C 180,E1 -12102.779,E2 -12102.779} C_VEL
LIN {X 0,Y 382.996,Z 287.077,A -85,B 0,C 180,E1 -12105.789,E2 -12105.789} C_VEL
LIN {X 0,Y 382.987,Z 287.093,A -85,B 0,C 180,E1 -12108.796,E2 -12108.796} C_VEL
LIN {X 0,Y 382.999,Z 287.065,A -85,B 0,C 180,E1 -12112.097,E2 -12112.097} C_VEL
LIN {X 0,Y 383.016,Z 287.172,A -85,B 0,C 180,E1 -12112.757,E2 -12112.757} C_VEL
LIN {X 0,Y 383.545,Z 289.028,A -85,B 0,C 180,E1 -12113.079,E2 -12113.079} C_VEL
LIN {X 0,Y 392.158,Z 303.726,A -85,B 0,C 180,E1 -12114.353,E2 -12114.353} C_VEL
LIN {X 0,Y 402.45,Z 323.379,A -85,B 0,C 180,E1 -12115.823,E2 -12115.823} C_VEL
LIN {X 0,Y 406.858,Z 332.797,A -85,B 0,C 180,E1 -12116.444,E2 -12116.444} C_VEL
LIN {X 0,Y 402.667,Z 492.254,A -85,B 0,C 180,E1 -12119.374,E2 -12119.374} C_VEL
LIN {X 0,Y 401.812,Z 507.803,A -85,B 0,C 180,E1 -12119.811,E2 -12119.811} C_VEL
LIN {X 0,Y 400.665,Z 523.597,A -85,B 0,C 180,E1 -12120.44,E2 -12120.44} C_VEL
LIN {X 0,Y 399.174,Z 539.178,A -85,B 0,C 180,E1 -12121.258,E2 -12121.258} C_VEL
LIN {X 0,Y 397.361,Z 554.983,A -85,B 0,C 180,E1 -12122.321,E2 -12122.321} C_VEL
LIN {X 0,Y 395.542,Z 569.043,A -85,B 0,C 180,E1 -12123.486,E2 -12123.486} C_VEL
LIN {X 0,Y 393.459,Z 583.259,A -85,B 0,C 180,E1 -12124.899,E2 -12124.899} C_VEL
LIN {X 0,Y 391.457,Z 596.187,A -85,B 0,C 180,E1 -12126.435,E2 -12126.435} C_VEL
LIN {X 0,Y 389.651,Z 607.457,A -85,B 0,C 180,E1 -12128.022,E2 -12128.022} C_VEL
LIN {X 0,Y 387.75,Z 618.569,A -85,B 0,C 180,E1 -12129.856,E2 -12129.856} C_VEL
LIN {X 0,Y 386.094,Z 629.309,A -85,B 0,C 180,E1 -12131.974,E2 -12131.974} C_VEL
LIN {X 0,Y 384.669,Z 638.327,A -85,B 0,C 180,E1 -12134.094,E2 -12134.094} C_VEL
LIN {X 0,Y 383.566,Z 645.859,A -85,B 0,C 180,E1 -12136.22,E2 -12136.22} C_VEL
LIN {X 0,Y 382.805,Z 652.017,A -85,B 0,C 180,E1 -12138.349,E2 -12138.349} C_VEL
LIN {X 0,Y 382.266,Z 657.063,A -85,B 0,C 180,E1 -12140.476,E2 -12140.476} C_VEL
LIN {X 0,Y 381.933,Z 661.103,A -85,B 0,C 180,E1 -12142.694,E2 -12142.694} C_VEL
LIN {X 0,Y 381.153,Z 662.431,A -85,B 0,C 180,E1 -12143.553,E2 -12143.553} C_VEL
LIN {X 0,Y 378.134,Z 664.268,A -85,B 0,C 180,E1 -12144.952,E2 -12144.952} C_VEL
LIN {X 0,Y 375.639,Z 665.444,A -85,B 0,C 180,E1 -12146.09,E2 -12146.09} C_VEL
LIN {X 0,Y 374.523,Z 666.242,A -85,B 0,C 180,E1 -12147.128,E2 -12147.128} C_VEL
LIN {X 0,Y 374.504,Z 666.26,A -85,B 0,C 180,E1 -12147.279,E2 -12147.279} C_VEL
LIN {X 0,Y 374.541,Z 666.949,A -85,B 0,C 180,E1 -12148.925,E2 -12148.925} C_VEL
LIN {X 0,Y 374.541,Z 666.964,A -85,B 0,C 180,E1 -12151.075,E2 -12151.075} C_VEL
LIN {X 0,Y 374.51,Z 666.057,A -85,B 0,C 180,E1 -12153.227,E2 -12153.227} C_VEL
LIN {X 0,Y 374.678,Z 664.178,A -85,B 0,C 180,E1 -12155.381,E2 -12155.381} C_VEL
LIN {X 0,Y 374.866,Z 661.333,A -85,B 0,C 180,E1 -12157.541,E2 -12157.541} C_VEL
LIN {X 0,Y 375.216,Z 657.459,A -85,B 0,C 180,E1 -12159.705,E2 -12159.705} C_VEL
LIN {X 0,Y 375.795,Z 652.478,A -85,B 0,C 180,E1 -12161.871,E2 -12161.871} C_VEL
LIN {X 0,Y 376.635,Z 646.385,A -85,B 0,C 180,E1 -12164.039,E2 -12164.039} C_VEL
LIN {X 0,Y 377.908,Z 637.898,A -85,B 0,C 180,E1 -12166.475,E2 -12166.475} C_VEL
LIN {X 0,Y 379.426,Z 628.906,A -85,B 0,C 180,E1 -12168.594,E2 -12168.594} C_VEL
LIN {X 0,Y 380.972,Z 619.304,A -85,B 0,C 180,E1 -12170.518,E2 -12170.518} C_VEL
LIN {X 0,Y 382.943,Z 608.298,A -85,B 0,C 180,E1 -12172.384,E2 -12172.384} C_VEL
LIN {X 0,Y 384.994,Z 596.221,A -85,B 0,C 180,E1 -12174.113,E2 -12174.113} C_VEL
LIN {X 0,Y 387.151,Z 583.123,A -85,B 0,C 180,E1 -12175.684,E2 -12175.684} C_VEL
LIN {X 0,Y 389.12,Z 570.251,A -85,B 0,C 180,E1 -12176.987,E2 -12176.987} C_VEL
LIN {X 0,Y 390.929,Z 556.286,A -85,B 0,C 180,E1 -12178.187,E2 -12178.187} C_VEL
LIN {X 0,Y 392.921,Z 539.827,A -85,B 0,C 180,E1 -12179.317,E2 -12179.317} C_VEL
LIN {X 0,Y 394.644,Z 523.016,A -85,B 0,C 180,E1 -12180.204,E2 -12180.204} C_VEL
LIN {X 0,Y 395.789,Z 506.896,A -85,B 0,C 180,E1 -12180.846,E2 -12180.846} C_VEL
LIN {X 0,Y 396.693,Z 490.299,A -85,B 0,C 180,E1 -12181.294,E2 -12181.294} C_VEL
LIN {X 0,Y 400.904,Z 335.756,A -85,B 0,C 180,E1 -12184.169,E2 -12184.169} C_VEL
LIN {X 0,Y 400.597,Z 334.006,A -85,B 0,C 180,E1 -12184.236,E2 -12184.236} C_VEL
LIN {X 0,Y 391.806,Z 316.394,A -85,B 0,C 180,E1 -12185.51,E2 -12185.51} C_VEL
LIN {X 0,Y 382.395,Z 299.438,A -85,B 0,C 180,E1 -12186.919,E2 -12186.919} C_VEL
LIN {X 0,Y 377.391,Z 291.375,A -85,B 0,C 180,E1 -12187.686,E2 -12187.686} C_VEL
LIN {X 0,Y 376.131,Z 288.886,A -85,B 0,C 180,E1 -12187.905,E2 -12187.905} C_VEL
LIN {X 0,Y 375.962,Z 287.959,A -85,B 0,C 180,E1 -12188.088,E2 -12188.088} C_VEL
LIN {X 0,Y 375.939,Z 287.969,A -85,B 0,C 180,E1 -12190.867,E2 -12190.867} C_VEL
LIN {X 0,Y 375.929,Z 287.972,A -85,B 0,C 180,E1 -12193.765,E2 -12193.765} C_VEL
LIN {X 0,Y 375.932,Z 287.968,A -85,B 0,C 180,E1 -12196.81,E2 -12196.81} C_VEL
LIN {X 0,Y 375.96,Z 287.965,A -85,B 0,C 180,E1 -12200.537,E2 -12200.537} C_VEL
LIN {X 0,Y 375.962,Z 287.956,A -85,B 0,C 180,E1 -12203.495,E2 -12203.495} C_VEL
LIN {X 0,Y 375.958,Z 287.963,A -85,B 0,C 180,E1 -12205.888,E2 -12205.888} C_VEL
LIN {X 0,Y 375.963,Z 287.966,A -85,B 0,C 180,E1 -12209.687,E2 -12209.687} C_VEL
LIN {X 0,Y 376.018,Z 287.947,A -85,B 0,C 180,E1 -12213.348,E2 -12213.348} C_VEL
LIN {X 0,Y 375.994,Z 287.948,A -85,B 0,C 180,E1 -12216.888,E2 -12216.888} C_VEL
LIN {X 0,Y 375.998,Z 287.959,A -85,B 0,C 180,E1 -12220.339,E2 -12220.339} C_VEL
LIN {X 0,Y 376.026,Z 287.933,A -85,B 0,C 180,E1 -12223.719,E2 -12223.719} C_VEL
LIN {X 0,Y 376.101,Z 287.951,A -85,B 0,C 180,E1 -12227.042,E2 -12227.042} C_VEL
LIN {X 0,Y 376.116,Z 287.922,A -85,B 0,C 180,E1 -12230.318,E2 -12230.318} C_VEL
LIN {X 0,Y 376.228,Z 287.925,A -85,B 0,C 180,E1 -12232.486,E2 -12232.486} C_VEL
LIN {X 0,Y 376.169,Z 287.941,A -85,B 0,C 180,E1 -12234.64,E2 -12234.64} C_VEL
LIN {X 0,Y 376.349,Z 287.896,A -85,B 0,C 180,E1 -12237.859,E2 -12237.859} C_VEL
LIN {X 0,Y 376.486,Z 287.898,A -85,B 0,C 180,E1 -12240,E2 -12240} C_VEL
LIN {X 0,Y 376.185,Z 287.914,A -85,B 0,C 180,E1 -12243.213,E2 -12243.213} C_VEL
LIN {X 0,Y 376.244,Z 287.927,A -85,B 0,C 180,E1 -12246.435,E2 -12246.435} C_VEL
LIN {X 0,Y 376.203,Z 287.931,A -85,B 0,C 180,E1 -12248.595,E2 -12248.595} C_VEL
LIN {X 0,Y 376.047,Z 287.945,A -85,B 0,C 180,E1 -12251.863,E2 -12251.863} C_VEL
LIN {X 0,Y 376.055,Z 287.951,A -85,B 0,C 180,E1 -12255.167,E2 -12255.167} C_VEL
LIN {X 0,Y 376.021,Z 287.955,A -85,B 0,C 180,E1 -12258.526,E2 -12258.526} C_VEL
LIN {X 0,Y 375.96,Z 287.964,A -85,B 0,C 180,E1 -12261.954,E2 -12261.954} C_VEL
LIN {X 0,Y 376.004,Z 287.964,A -85,B 0,C 180,E1 -12265.461,E2 -12265.461} C_VEL
LIN {X 0,Y 375.967,Z 287.969,A -85,B 0,C 180,E1 -12269.079,E2 -12269.079} C_VEL
LIN {X 0,Y 375.946,Z 287.97,A -85,B 0,C 180,E1 -12272.829,E2 -12272.829} C_VEL
LIN {X 0,Y 375.955,Z 287.967,A -85,B 0,C 180,E1 -12275.415,E2 -12275.415} C_VEL
LIN {X 0,Y 375.972,Z 287.97,A -85,B 0,C 180,E1 -12278.271,E2 -12278.271} C_VEL
LIN {X 0,Y 375.931,Z 287.974,A -85,B 0,C 180,E1 -12281.601,E2 -12281.601} C_VEL
LIN {X 0,Y 375.926,Z 287.975,A -85,B 0,C 180,E1 -12285.268,E2 -12285.268} C_VEL
LIN {X 0,Y 375.979,Z 287.967,A -85,B 0,C 180,E1 -12289.138,E2 -12289.138} C_VEL
LIN {X 0,Y 376.007,Z 288.15,A -85,B 0,C 180,E1 -12289.345,E2 -12289.345} C_VEL
LIN {X 0,Y 381.456,Z 303.664,A -85,B 0,C 180,E1 -12292.395,E2 -12292.395} C_VEL
LIN {X 0,Y 382.517,Z 306.496,A -85,B 0,C 180,E1 -12292.891,E2 -12292.891} C_VEL
LIN {X 0,Y 391.602,Z 323.664,A -85,B 0,C 180,E1 -12294.264,E2 -12294.264} C_VEL
LIN {X 0,Y 399.229,Z 339.669,A -85,B 0,C 180,E1 -12295.385,E2 -12295.385} C_VEL
LIN {X 0,Y 400.673,Z 349.58,A -85,B 0,C 180,E1 -12295.737,E2 -12295.737} C_VEL
LIN {X 0,Y 396.18,Z 513.809,A -85,B 0,C 180,E1 -12298.797,E2 -12298.797} C_VEL
LIN {X 0,Y 395.033,Z 530.198,A -85,B 0,C 180,E1 -12299.274,E2 -12299.274} C_VEL
LIN {X 0,Y 393.643,Z 546.03,A -85,B 0,C 180,E1 -12299.933,E2 -12299.933} C_VEL
LIN {X 0,Y 391.994,Z 561.212,A -85,B 0,C 180,E1 -12300.754,E2 -12300.754} C_VEL
LIN {X 0,Y 390.145,Z 576.186,A -85,B 0,C 180,E1 -12301.78,E2 -12301.78} C_VEL
LIN {X 0,Y 387.931,Z 591.459,A -85,B 0,C 180,E1 -12303.069,E2 -12303.069} C_VEL
LIN {X 0,Y 385.869,Z 604.277,A -85,B 0,C 180,E1 -12304.37,E2 -12304.37} C_VEL
LIN {X 0,Y 383.763,Z 617.421,A -85,B 0,C 180,E1 -12305.954,E2 -12305.954} C_VEL
LIN {X 0,Y 381.924,Z 628.662,A -85,B 0,C 180,E1 -12307.553,E2 -12307.553} C_VEL
LIN {X 0,Y 380.01,Z 639.873,A -85,B 0,C 180,E1 -12309.428,E2 -12309.428} C_VEL
LIN {X 0,Y 378.238,Z 650.745,A -85,B 0,C 180,E1 -12311.587,E2 -12311.587} C_VEL
LIN {X 0,Y 376.909,Z 659.89,A -85,B 0,C 180,E1 -12313.758,E2 -12313.758} C_VEL
LIN {X 0,Y 375.938,Z 667.558,A -85,B 0,C 180,E1 -12315.935,E2 -12315.935} C_VEL
LIN {X 0,Y 375.249,Z 673.82,A -85,B 0,C 180,E1 -12318.111,E2 -12318.111} C_VEL
LIN {X 0,Y 374.786,Z 678.956,A -85,B 0,C 180,E1 -12320.284,E2 -12320.284} C_VEL
LIN {X 0,Y 374.618,Z 682.952,A -85,B 0,C 180,E1 -12322.454,E2 -12322.454} C_VEL
LIN {X 0,Y 374.495,Z 685.909,A -85,B 0,C 180,E1 -12324.616,E2 -12324.616} C_VEL
LIN {X 0,Y 374.441,Z 687.856,A -85,B 0,C 180,E1 -12326.772,E2 -12326.772} C_VEL
LIN {X 0,Y 374.512,Z 688.824,A -85,B 0,C 180,E1 -12328.925,E2 -12328.925} C_VEL
LIN {X 0,Y 374.512,Z 688.822,A -85,B 0,C 180,E1 -12331.075,E2 -12331.075} C_VEL
LIN {X 0,Y 374.441,Z 687.85,A -85,B 0,C 180,E1 -12333.228,E2 -12333.228} C_VEL
LIN {X 0,Y 374.495,Z 685.9,A -85,B 0,C 180,E1 -12335.384,E2 -12335.384} C_VEL
LIN {X 0,Y 374.618,Z 682.941,A -85,B 0,C 180,E1 -12337.546,E2 -12337.546} C_VEL
LIN {X 0,Y 374.786,Z 678.944,A -85,B 0,C 180,E1 -12339.716,E2 -12339.716} C_VEL
LIN {X 0,Y 375.248,Z 673.802,A -85,B 0,C 180,E1 -12341.889,E2 -12341.889} C_VEL
LIN {X 0,Y 375.936,Z 667.531,A -85,B 0,C 180,E1 -12344.065,E2 -12344.065} C_VEL
LIN {X 0,Y 377.083,Z 658.84,A -85,B 0,C 180,E1 -12346.513,E2 -12346.513} C_VEL
LIN {X 0,Y 378.519,Z 649.144,A -85,B 0,C 180,E1 -12348.752,E2 -12348.752} C_VEL
LIN {X 0,Y 379.999,Z 639.823,A -85,B 0,C 180,E1 -12350.573,E2 -12350.573} C_VEL
LIN {X 0,Y 381.973,Z 628.599,A -85,B 0,C 180,E1 -12352.444,E2 -12352.444} C_VEL
LIN {X 0,Y 383.914,Z 616.367,A -85,B 0,C 180,E1 -12354.18,E2 -12354.18} C_VEL
LIN {X 0,Y 386.082,Z 603.01,A -85,B 0,C 180,E1 -12355.76,E2 -12355.76} C_VEL
LIN {X 0,Y 388.236,Z 589.311,A -85,B 0,C 180,E1 -12357.115,E2 -12357.115} C_VEL
LIN {X 0,Y 390.138,Z 576.04,A -85,B 0,C 180,E1 -12358.221,E2 -12358.221} C_VEL
LIN {X 0,Y 392.133,Z 560.044,A -85,B 0,C 180,E1 -12359.308,E2 -12359.308} C_VEL
LIN {X 0,Y 393.773,Z 544.517,A -85,B 0,C 180,E1 -12360.13,E2 -12360.13} C_VEL
LIN {X 0,Y 395.095,Z 528.983,A -85,B 0,C 180,E1 -12360.757,E2 -12360.757} C_VEL
LIN {X 0,Y 396.163,Z 513.465,A -85,B 0,C 180,E1 -12361.2,E2 -12361.2} C_VEL
LIN {X 0,Y 400.287,Z 360.827,A -85,B 0,C 180,E1 -12364.049,E2 -12364.049} C_VEL
LIN {X 0,Y 400.544,Z 347.817,A -85,B 0,C 180,E1 -12364.3,E2 -12364.3} C_VEL
LIN {X 0,Y 399.056,Z 339.314,A -85,B 0,C 180,E1 -12364.626,E2 -12364.626} C_VEL
LIN {X 0,Y 390.889,Z 322.312,A -85,B 0,C 180,E1 -12365.825,E2 -12365.825} C_VEL
LIN {X 0,Y 382.25,Z 305.884,A -85,B 0,C 180,E1 -12367.165,E2 -12367.165} C_VEL
LIN {X 0,Y 376.882,Z 290.619,A -85,B 0,C 180,E1 -12370.133,E2 -12370.133} C_VEL
LIN {X 0,Y 375.945,Z 287.967,A -85,B 0,C 180,E1 -12370.71,E2 -12370.71} C_VEL
LIN {X 0,Y 375.929,Z 287.968,A -85,B 0,C 180,E1 -12373.766,E2 -12373.766} C_VEL
LIN {X 0,Y 375.931,Z 287.965,A -85,B 0,C 180,E1 -12376.811,E2 -12376.811} C_VEL
LIN {X 0,Y 375.959,Z 287.958,A -85,B 0,C 180,E1 -12380.537,E2 -12380.537} C_VEL
LIN {X 0,Y 375.961,Z 287.964,A -85,B 0,C 180,E1 -12383.496,E2 -12383.496} C_VEL
LIN {X 0,Y 375.957,Z 287.964,A -85,B 0,C 180,E1 -12385.889,E2 -12385.889} C_VEL
LIN {X 0,Y 375.962,Z 287.961,A -85,B 0,C 180,E1 -12389.687,E2 -12389.687} C_VEL
LIN {X 0,Y 375.994,Z 287.959,A -85,B 0,C 180,E1 -12392.141,E2 -12392.141} C_VEL
LIN {X 0,Y 376.004,Z 287.961,A -85,B 0,C 180,E1 -12394.539,E2 -12394.539} C_VEL
LIN {X 0,Y 375.966,Z 287.961,A -85,B 0,C 180,E1 -12398.046,E2 -12398.046} C_VEL
LIN {X 0,Y 376.021,Z 287.946,A -85,B 0,C 180,E1 -12401.474,E2 -12401.474} C_VEL
LIN {X 0,Y 376.056,Z 287.942,A -85,B 0,C 180,E1 -12404.833,E2 -12404.833} C_VEL
LIN {X 0,Y 376.048,Z 287.945,A -85,B 0,C 180,E1 -12408.137,E2 -12408.137} C_VEL
LIN {X 0,Y 376.217,Z 287.922,A -85,B 0,C 180,E1 -12411.919,E2 -12411.919} C_VEL
LIN {X 0,Y 376.169,Z 287.919,A -85,B 0,C 180,E1 -12414.64,E2 -12414.64} C_VEL
LIN {X 0,Y 376.352,Z 287.914,A -85,B 0,C 180,E1 -12417.86,E2 -12417.86} C_VEL
LIN {X 0,Y 376.485,Z 287.877,A -85,B 0,C 180,E1 -12420,E2 -12420} C_VEL
LIN {X 0,Y 376.184,Z 287.932,A -85,B 0,C 180,E1 -12423.213,E2 -12423.213} C_VEL
LIN {X 0,Y 376.229,Z 287.918,A -85,B 0,C 180,E1 -12426.553,E2 -12426.553} C_VEL
LIN {X 0,Y 376.117,Z 287.932,A -85,B 0,C 180,E1 -12429.682,E2 -12429.682} C_VEL
LIN {X 0,Y 376.088,Z 287.938,A -85,B 0,C 180,E1 -12433.658,E2 -12433.658} C_VEL
LIN {X 0,Y 376.042,Z 287.954,A -85,B 0,C 180,E1 -12437.607,E2 -12437.607} C_VEL
LIN {X 0,Y 375.977,Z 287.945,A -85,B 0,C 180,E1 -12440.832,E2 -12440.832} C_VEL
LIN {X 0,Y 375.992,Z 287.959,A -85,B 0,C 180,E1 -12444.282,E2 -12444.282} C_VEL
LIN {X 0,Y 376.018,Z 287.946,A -85,B 0,C 180,E1 -12446.652,E2 -12446.652} C_VEL
LIN {X 0,Y 375.963,Z 287.964,A -85,B 0,C 180,E1 -12450.313,E2 -12450.313} C_VEL
LIN {X 0,Y 375.959,Z 287.964,A -85,B 0,C 180,E1 -12454.112,E2 -12454.112} C_VEL
LIN {X 0,Y 375.952,Z 287.958,A -85,B 0,C 180,E1 -12456.741,E2 -12456.741} C_VEL
LIN {X 0,Y 375.987,Z 287.959,A -85,B 0,C 180,E1 -12459.971,E2 -12459.971} C_VEL
LIN {X 0,Y 375.929,Z 287.968,A -85,B 0,C 180,E1 -12463.766,E2 -12463.766} C_VEL
LIN {X 0,Y 375.933,Z 287.963,A -85,B 0,C 180,E1 -12466.811,E2 -12466.811} C_VEL
LIN {X 0,Y 375.962,Z 287.969,A -85,B 0,C 180,E1 -12470.538,E2 -12470.538} C_VEL
LIN {X 0,Y 375.993,Z 288.06,A -85,B 0,C 180,E1 -12472.047,E2 -12472.047} C_VEL
LIN {X 0,Y 376.223,Z 289.152,A -85,B 0,C 180,E1 -12472.233,E2 -12472.233} C_VEL
LIN {X 0,Y 377.676,Z 291.732,A -85,B 0,C 180,E1 -12472.465,E2 -12472.465} C_VEL
LIN {X 0,Y 384.425,Z 302.965,A -85,B 0,C 180,E1 -12473.498,E2 -12473.498} C_VEL
LIN {X 0,Y 393.834,Z 320.341,A -85,B 0,C 180,E1 -12474.894,E2 -12474.894} C_VEL
LIN {X 0,Y 400.901,Z 334.698,A -85,B 0,C 180,E1 -12475.912,E2 -12475.912} C_VEL
LIN {X 0,Y 396.585,Z 492.717,A -85,B 0,C 180,E1 -12478.858,E2 -12478.858} C_VEL
LIN {X 0,Y 395.635,Z 508.937,A -85,B 0,C 180,E1 -12479.326,E2 -12479.326} C_VEL
LIN {X 0,Y 394.391,Z 525.109,A -85,B 0,C 180,E1 -12479.996,E2 -12479.996} C_VEL
LIN {X 0,Y 392.853,Z 540.437,A -85,B 0,C 180,E1 -12480.824,E2 -12480.824} C_VEL
LIN {X 0,Y 390.984,Z 555.883,A -85,B 0,C 180,E1 -12481.887,E2 -12481.887} C_VEL
LIN {X 0,Y 388.959,Z 570.677,A -85,B 0,C 180,E1 -12483.146,E2 -12483.146} C_VEL
LIN {X 0,Y 386.816,Z 584.639,A -85,B 0,C 180,E1 -12484.581,E2 -12484.581} C_VEL
LIN {X 0,Y 384.554,Z 598.481,A -85,B 0,C 180,E1 -12486.293,E2 -12486.293} C_VEL
LIN {X 0,Y 382.411,Z 611.024,A -85,B 0,C 180,E1 -12488.151,E2 -12488.151} C_VEL
LIN {X 0,Y 380.562,Z 621.703,A -85,B 0,C 180,E1 -12490.023,E2 -12490.023} C_VEL
LIN {X 0,Y 378.865,Z 631.961,A -85,B 0,C 180,E1 -12492.177,E2 -12492.177} C_VEL
LIN {X 0,Y 377.468,Z 640.533,A -85,B 0,C 180,E1 -12494.337,E2 -12494.337} C_VEL
LIN {X 0,Y 376.362,Z 647.809,A -85,B 0,C 180,E1 -12496.538,E2 -12496.538} C_VEL
LIN {X 0,Y 375.624,Z 653.634,A -85,B 0,C 180,E1 -12498.67,E2 -12498.67} C_VEL
LIN {X 0,Y 375.02,Z 659.376,A -85,B 0,C 180,E1 -12501.378,E2 -12501.378} C_VEL
LIN {X 0,Y 374.771,Z 662.907,A -85,B 0,C 180,E1 -12503.668,E2 -12503.668} C_VEL
LIN {X 0,Y 374.582,Z 665.182,A -85,B 0,C 180,E1 -12505.696,E2 -12505.696} C_VEL
LIN {X 0,Y 374.504,Z 666.26,A -85,B 0,C 180,E1 -12507.279,E2 -12507.279} C_VEL
LIN {X 0,Y 373.844,Z 666.747,A -85,B 0,C 180,E1 -12508.174,E2 -12508.174} C_VEL
LIN {X 0,Y 370.961,Z 667.158,A -85,B 0,C 180,E1 -12509.632,E2 -12509.632} C_VEL
LIN {X 0,Y 368.525,Z 667.18,A -85,B 0,C 180,E1 -12510.813,E2 -12510.813} C_VEL
LIN {X 0,Y 367.498,Z 667.02,A -85,B 0,C 180,E1 -12511.726,E2 -12511.726} C_VEL
LIN {X 0,Y 367.425,Z 666.872,A -85,B 0,C 180,E1 -12512.034,E2 -12512.034} C_VEL
LIN {X 0,Y 367.514,Z 665.476,A -85,B 0,C 180,E1 -12514.387,E2 -12514.387} C_VEL
LIN {X 0,Y 367.693,Z 663.075,A -85,B 0,C 180,E1 -12516.585,E2 -12516.585} C_VEL
LIN {X 0,Y 367.968,Z 659.766,A -85,B 0,C 180,E1 -12518.789,E2 -12518.789} C_VEL
LIN {X 0,Y 368.592,Z 654.08,A -85,B 0,C 180,E1 -12521.549,E2 -12521.549} C_VEL
LIN {X 0,Y 369.674,Z 646.593,A -85,B 0,C 180,E1 -12524.309,E2 -12524.309} C_VEL
LIN {X 0,Y 371.05,Z 638.105,A -85,B 0,C 180,E1 -12526.789,E2 -12526.789} C_VEL
LIN {X 0,Y 372.628,Z 629.096,A -85,B 0,C 180,E1 -12528.95,E2 -12528.95} C_VEL
LIN {X 0,Y 374.266,Z 619.51,A -85,B 0,C 180,E1 -12530.903,E2 -12530.903} C_VEL
LIN {X 0,Y 376.336,Z 608.504,A -85,B 0,C 180,E1 -12532.799,E2 -12532.799} C_VEL
LIN {X 0,Y 378.381,Z 596.981,A -85,B 0,C 180,E1 -12534.478,E2 -12534.478} C_VEL
LIN {X 0,Y 380.525,Z 584.495,A -85,B 0,C 180,E1 -12536.017,E2 -12536.017} C_VEL
LIN {X 0,Y 382.569,Z 571.874,A -85,B 0,C 180,E1 -12537.339,E2 -12537.339} C_VEL
LIN {X 0,Y 384.609,Z 557.055,A -85,B 0,C 180,E1 -12538.643,E2 -12538.643} C_VEL
LIN {X 0,Y 386.493,Z 542.024,A -85,B 0,C 180,E1 -12539.703,E2 -12539.703} C_VEL
LIN {X 0,Y 388.167,Z 527.105,A -85,B 0,C 180,E1 -12540.536,E2 -12540.536} C_VEL
LIN {X 0,Y 389.443,Z 510.747,A -85,B 0,C 180,E1 -12541.254,E2 -12541.254} C_VEL
LIN {X 0,Y 390.512,Z 494.84,A -85,B 0,C 180,E1 -12541.737,E2 -12541.737} C_VEL
LIN {X 0,Y 394.957,Z 336.795,A -85,B 0,C 180,E1 -12544.738,E2 -12544.738} C_VEL
LIN {X 0,Y 384.888,Z 316.704,A -85,B 0,C 180,E1 -12546.246,E2 -12546.246} C_VEL
LIN {X 0,Y 375.347,Z 299.918,A -85,B 0,C 180,E1 -12547.726,E2 -12547.726} C_VEL
LIN {X 0,Y 371.504,Z 293.635,A -85,B 0,C 180,E1 -12548.341,E2 -12548.341} C_VEL
LIN {X 0,Y 369.427,Z 290.737,A -85,B 0,C 180,E1 -12548.669,E2 -12548.669} C_VEL
LIN {X 0,Y 368.933,Z 288.91,A -85,B 0,C 180,E1 -12548.822,E2 -12548.822} C_VEL
LIN {X 0,Y 368.88,Z 288.842,A -85,B 0,C 180,E1 -12552.009,E2 -12552.009} C_VEL
LIN {X 0,Y 368.878,Z 288.84,A -85,B 0,C 180,E1 -12555.175,E2 -12555.175} C_VEL
LIN {X 0,Y 368.881,Z 288.843,A -85,B 0,C 180,E1 -12558.177,E2 -12558.177} C_VEL
LIN {X 0,Y 368.906,Z 288.844,A -85,B 0,C 180,E1 -12561.36,E2 -12561.36} C_VEL
LIN {X 0,Y 368.935,Z 288.844,A -85,B 0,C 180,E1 -12565.146,E2 -12565.146} C_VEL
LIN {X 0,Y 368.927,Z 288.839,A -85,B 0,C 180,E1 -12569.046,E2 -12569.046} C_VEL
LIN {X 0,Y 368.961,Z 288.82,A -85,B 0,C 180,E1 -12572.796,E2 -12572.796} C_VEL
LIN {X 0,Y 368.943,Z 288.836,A -85,B 0,C 180,E1 -12576.113,E2 -12576.113} C_VEL
LIN {X 0,Y 368.936,Z 288.839,A -85,B 0,C 180,E1 -12579.947,E2 -12579.947} C_VEL
LIN {X 0,Y 368.973,Z 288.813,A -85,B 0,C 180,E1 -12583.398,E2 -12583.398} C_VEL
LIN {X 0,Y 369.055,Z 288.826,A -85,B 0,C 180,E1 -12586.79,E2 -12586.79} C_VEL
LIN {X 0,Y 369.065,Z 288.8,A -85,B 0,C 180,E1 -12590.132,E2 -12590.132} C_VEL
LIN {X 0,Y 369.186,Z 288.802,A -85,B 0,C 180,E1 -12592.342,E2 -12592.342} C_VEL
LIN {X 0,Y 369.142,Z 288.816,A -85,B 0,C 180,E1 -12594.537,E2 -12594.537} C_VEL
LIN {X 0,Y 369.314,Z 288.772,A -85,B 0,C 180,E1 -12597.819,E2 -12597.819} C_VEL
LIN {X 0,Y 369.456,Z 288.774,A -85,B 0,C 180,E1 -12600,E2 -12600} C_VEL
LIN {X 0,Y 369.316,Z 288.788,A -85,B 0,C 180,E1 -12602.181,E2 -12602.181} C_VEL
LIN {X 0,Y 369.206,Z 288.804,A -85,B 0,C 180,E1 -12606.558,E2 -12606.558} C_VEL
LIN {X 0,Y 369.135,Z 288.808,A -85,B 0,C 180,E1 -12608.761,E2 -12608.761} C_VEL
LIN {X 0,Y 369.002,Z 288.823,A -85,B 0,C 180,E1 -12612.093,E2 -12612.093} C_VEL
LIN {X 0,Y 368.995,Z 288.83,A -85,B 0,C 180,E1 -12615.465,E2 -12615.465} C_VEL
LIN {X 0,Y 368.98,Z 288.834,A -85,B 0,C 180,E1 -12618.893,E2 -12618.893} C_VEL
LIN {X 0,Y 368.929,Z 288.842,A -85,B 0,C 180,E1 -12622.395,E2 -12622.395} C_VEL
LIN {X 0,Y 368.997,Z 288.836,A -85,B 0,C 180,E1 -12625.98,E2 -12625.98} C_VEL
LIN {X 0,Y 368.958,Z 288.846,A -85,B 0,C 180,E1 -12628.812,E2 -12628.812} C_VEL
LIN {X 0,Y 368.895,Z 288.852,A -85,B 0,C 180,E1 -12632.238,E2 -12632.238} C_VEL
LIN {X 0,Y 368.926,Z 288.845,A -85,B 0,C 180,E1 -12635.002,E2 -12635.002} C_VEL
LIN {X 0,Y 368.907,Z 288.851,A -85,B 0,C 180,E1 -12638.641,E2 -12638.641} C_VEL
LIN {X 0,Y 368.878,Z 288.854,A -85,B 0,C 180,E1 -12642.009,E2 -12642.009} C_VEL
LIN {X 0,Y 368.879,Z 288.853,A -85,B 0,C 180,E1 -12645.176,E2 -12645.176} C_VEL
LIN {X 0,Y 368.918,Z 288.942,A -85,B 0,C 180,E1 -12648.565,E2 -12648.565} C_VEL
LIN {X 0,Y 374.483,Z 304.482,A -85,B 0,C 180,E1 -12651.734,E2 -12651.734} C_VEL
LIN {X 0,Y 375.044,Z 306.081,A -85,B 0,C 180,E1 -12652.019,E2 -12652.019} C_VEL
LIN {X 0,Y 384.294,Z 323.1,A -85,B 0,C 180,E1 -12653.468,E2 -12653.468} C_VEL
LIN {X 0,Y 393.584,Z 342.412,A -85,B 0,C 180,E1 -12654.879,E2 -12654.879} C_VEL
LIN {X 0,Y 394.777,Z 349.776,A -85,B 0,C 180,E1 -12655.16,E2 -12655.16} C_VEL
LIN {X 0,Y 390.259,Z 509.387,A -85,B 0,C 180,E1 -12658.163,E2 -12658.163} C_VEL
LIN {X 0,Y 389.299,Z 525.415,A -85,B 0,C 180,E1 -12658.582,E2 -12658.582} C_VEL
LIN {X 0,Y 387.984,Z 541.163,A -85,B 0,C 180,E1 -12659.184,E2 -12659.184} C_VEL
LIN {X 0,Y 386.343,Z 556.673,A -85,B 0,C 180,E1 -12659.983,E2 -12659.983} C_VEL
LIN {X 0,Y 384.308,Z 572.439,A -85,B 0,C 180,E1 -12661.013,E2 -12661.013} C_VEL
LIN {X 0,Y 382.173,Z 587.482,A -85,B 0,C 180,E1 -12662.239,E2 -12662.239} C_VEL
LIN {X 0,Y 379.822,Z 601.713,A -85,B 0,C 180,E1 -12663.636,E2 -12663.636} C_VEL
LIN {X 0,Y 377.491,Z 615.202,A -85,B 0,C 180,E1 -12665.235,E2 -12665.235} C_VEL
LIN {X 0,Y 375.56,Z 626.66,A -85,B 0,C 180,E1 -12666.86,E2 -12666.86} C_VEL
LIN {X 0,Y 373.538,Z 638.169,A -85,B 0,C 180,E1 -12668.766,E2 -12668.766} C_VEL
LIN {X 0,Y 371.847,Z 648.052,A -85,B 0,C 180,E1 -12670.686,E2 -12670.686} C_VEL
LIN {X 0,Y 370.375,Z 657.561,A -85,B 0,C 180,E1 -12672.896,E2 -12672.896} C_VEL
LIN {X 0,Y 369.171,Z 665.521,A -85,B 0,C 180,E1 -12675.108,E2 -12675.108} C_VEL
LIN {X 0,Y 368.417,Z 672.172,A -85,B 0,C 180,E1 -12677.328,E2 -12677.328} C_VEL
LIN {X 0,Y 367.803,Z 677.569,A -85,B 0,C 180,E1 -12679.541,E2 -12679.541} C_VEL
LIN {X 0,Y 367.599,Z 680.908,A -85,B 0,C 180,E1 -12681.202,E2 -12681.202} C_VEL
LIN {X 0,Y 367.472,Z 685.117,A -85,B 0,C 180,E1 -12683.992,E2 -12683.992} C_VEL
LIN {X 0,Y 367.399,Z 686.833,A -85,B 0,C 180,E1 -12685.612,E2 -12685.612} C_VEL
LIN {X 0,Y 367.35,Z 688.24,A -85,B 0,C 180,E1 -12687.807,E2 -12687.807} C_VEL
LIN {X 0,Y 367.452,Z 688.772,A -85,B 0,C 180,E1 -12690,E2 -12690} C_VEL
LIN {X 0,Y 367.35,Z 688.236,A -85,B 0,C 180,E1 -12692.193,E2 -12692.193} C_VEL
LIN {X 0,Y 367.399,Z 686.825,A -85,B 0,C 180,E1 -12694.388,E2 -12694.388} C_VEL
LIN {X 0,Y 367.476,Z 684.328,A -85,B 0,C 180,E1 -12696.589,E2 -12696.589} C_VEL
LIN {X 0,Y 367.599,Z 680.895,A -85,B 0,C 180,E1 -12698.798,E2 -12698.798} C_VEL
LIN {X 0,Y 368.085,Z 675.028,A -85,B 0,C 180,E1 -12701.565,E2 -12701.565} C_VEL
LIN {X 0,Y 368.784,Z 668.815,A -85,B 0,C 180,E1 -12703.836,E2 -12703.836} C_VEL
LIN {X 0,Y 369.825,Z 660.663,A -85,B 0,C 180,E1 -12706.278,E2 -12706.278} C_VEL
LIN {X 0,Y 371.226,Z 651.736,A -85,B 0,C 180,E1 -12708.488,E2 -12708.488} C_VEL
LIN {X 0,Y 373.006,Z 641.107,A -85,B 0,C 180,E1 -12710.688,E2 -12710.688} C_VEL
LIN {X 0,Y 375.001,Z 630.123,A -85,B 0,C 180,E1 -12712.594,E2 -12712.594} C_VEL
LIN {X 0,Y 377.173,Z 617.135,A -85,B 0,C 180,E1 -12714.493,E2 -12714.493} C_VEL
LIN {X 0,Y 379.418,Z 603.976,A -85,B 0,C 180,E1 -12716.099,E2 -12716.099} C_VEL
LIN {X 0,Y 381.541,Z 591.134,A -85,B 0,C 180,E1 -12717.419,E2 -12717.419} C_VEL
LIN {X 0,Y 383.625,Z 577.507,A -85,B 0,C 180,E1 -12718.594,E2 -12718.594} C_VEL
LIN {X 0,Y 385.538,Z 562.822,A -85,B 0,C 180,E1 -12719.634,E2 -12719.634} C_VEL
LIN {X 0,Y 387.382,Z 546.907,A -85,B 0,C 180,E1 -12720.529,E2 -12720.529} C_VEL
LIN {X 0,Y 388.804,Z 531.518,A -85,B 0,C 180,E1 -12721.197,E2 -12721.197} C_VEL
LIN {X 0,Y 390.006,Z 515.087,A -85,B 0,C 180,E1 -12721.698,E2 -12721.698} C_VEL
LIN {X 0,Y 391.152,Z 474.581,A -85,B 0,C 180,E1 -12722.497,E2 -12722.497} C_VEL
LIN {X 0,Y 394.373,Z 362.549,A -85,B 0,C 180,E1 -12724.589,E2 -12724.589} C_VEL
LIN {X 0,Y 394.742,Z 349.472,A -85,B 0,C 180,E1 -12724.835,E2 -12724.835} C_VEL
LIN {X 0,Y 393.349,Z 341.895,A -85,B 0,C 180,E1 -12725.141,E2 -12725.141} C_VEL
LIN {X 0,Y 384.241,Z 323.05,A -85,B 0,C 180,E1 -12726.521,E2 -12726.521} C_VEL
LIN {X 0,Y 374.91,Z 305.861,A -85,B 0,C 180,E1 -12727.983,E2 -12727.983} C_VEL
LIN {X 0,Y 370.887,Z 294.236,A -85,B 0,C 180,E1 -12730.297,E2 -12730.297} C_VEL
LIN {X 0,Y 368.893,Z 288.847,A -85,B 0,C 180,E1 -12731.438,E2 -12731.438} C_VEL
LIN {X 0,Y 368.924,Z 288.842,A -85,B 0,C 180,E1 -12735.183,E2 -12735.183} C_VEL
LIN {X 0,Y 368.88,Z 288.84,A -85,B 0,C 180,E1 -12738.177,E2 -12738.177} C_VEL
LIN {X 0,Y 368.906,Z 288.843,A -85,B 0,C 180,E1 -12741.36,E2 -12741.36} C_VEL
LIN {X 0,Y 368.934,Z 288.835,A -85,B 0,C 180,E1 -12745.147,E2 -12745.147} C_VEL
LIN {X 0,Y 368.927,Z 288.842,A -85,B 0,C 180,E1 -12749.047,E2 -12749.047} C_VEL
LIN {X 0,Y 368.977,Z 288.836,A -85,B 0,C 180,E1 -12751.564,E2 -12751.564} C_VEL
LIN {X 0,Y 368.998,Z 288.833,A -85,B 0,C 180,E1 -12754.02,E2 -12754.02} C_VEL
LIN {X 0,Y 368.933,Z 288.839,A -85,B 0,C 180,E1 -12757.605,E2 -12757.605} C_VEL
LIN {X 0,Y 368.964,Z 288.818,A -85,B 0,C 180,E1 -12761.106,E2 -12761.106} C_VEL
LIN {X 0,Y 368.995,Z 288.827,A -85,B 0,C 180,E1 -12764.535,E2 -12764.535} C_VEL
LIN {X 0,Y 369.003,Z 288.818,A -85,B 0,C 180,E1 -12767.907,E2 -12767.907} C_VEL
LIN {X 0,Y 369.164,Z 288.801,A -85,B 0,C 180,E1 -12771.869,E2 -12771.869} C_VEL
LIN {X 0,Y 369.142,Z 288.793,A -85,B 0,C 180,E1 -12774.538,E2 -12774.538} C_VEL
LIN {X 0,Y 369.317,Z 288.791,A -85,B 0,C 180,E1 -12777.819,E2 -12777.819} C_VEL
LIN {X 0,Y 369.454,Z 288.752,A -85,B 0,C 180,E1 -12780,E2 -12780} C_VEL
LIN {X 0,Y 369.315,Z 288.777,A -85,B 0,C 180,E1 -12782.181,E2 -12782.181} C_VEL
LIN {X 0,Y 369.199,Z 288.792,A -85,B 0,C 180,E1 -12786.558,E2 -12786.558} C_VEL
LIN {X 0,Y 369.066,Z 288.813,A -85,B 0,C 180,E1 -12789.868,E2 -12789.868} C_VEL
LIN {X 0,Y 369.035,Z 288.816,A -85,B 0,C 180,E1 -12793.772,E2 -12793.772} C_VEL
LIN {X 0,Y 369,Z 288.831,A -85,B 0,C 180,E1 -12797.769,E2 -12797.769} C_VEL
LIN {X 0,Y 368.909,Z 288.82,A -85,B 0,C 180,E1 -12801.221,E2 -12801.221} C_VEL
LIN {X 0,Y 368.956,Z 288.84,A -85,B 0,C 180,E1 -12804.776,E2 -12804.776} C_VEL
LIN {X 0,Y 368.961,Z 288.817,A -85,B 0,C 180,E1 -12807.204,E2 -12807.204} C_VEL
LIN {X 0,Y 368.928,Z 288.843,A -85,B 0,C 180,E1 -12810.954,E2 -12810.954} C_VEL
LIN {X 0,Y 368.928,Z 288.839,A -85,B 0,C 180,E1 -12815.002,E2 -12815.002} C_VEL
LIN {X 0,Y 368.906,Z 288.827,A -85,B 0,C 180,E1 -12818.64,E2 -12818.64} C_VEL
LIN {X 0,Y 368.88,Z 288.832,A -85,B 0,C 180,E1 -12822.01,E2 -12822.01} C_VEL
LIN {X 0,Y 368.879,Z 288.839,A -85,B 0,C 180,E1 -12825.176,E2 -12825.176} C_VEL
LIN {X 0,Y 368.882,Z 288.848,A -85,B 0,C 180,E1 -12828.178,E2 -12828.178} C_VEL
LIN {X 0,Y 368.942,Z 289.003,A -85,B 0,C 180,E1 -12831.308,E2 -12831.308} C_VEL
LIN {X 0,Y 370.146,Z 292.019,A -85,B 0,C 180,E1 -12831.564,E2 -12831.564} C_VEL
LIN {X 0,Y 371.615,Z 293.927,A -85,B 0,C 180,E1 -12831.791,E2 -12831.791} C_VEL
LIN {X 0,Y 379.397,Z 306.911,A -85,B 0,C 180,E1 -12833.021,E2 -12833.021} C_VEL
LIN {X 0,Y 387.965,Z 322.728,A -85,B 0,C 180,E1 -12834.33,E2 -12834.33} C_VEL
LIN {X 0,Y 394.93,Z 336.882,A -85,B 0,C 180,E1 -12835.366,E2 -12835.366} C_VEL
LIN {X 0,Y 390.573,Z 492.067,A -85,B 0,C 180,E1 -12838.302,E2 -12838.302} C_VEL
LIN {X 0,Y 389.646,Z 508.242,A -85,B 0,C 180,E1 -12838.764,E2 -12838.764} C_VEL
LIN {X 0,Y 388.397,Z 524.029,A -85,B 0,C 180,E1 -12839.408,E2 -12839.408} C_VEL
LIN {X 0,Y 386.765,Z 539.609,A -85,B 0,C 180,E1 -12840.245,E2 -12840.245} C_VEL
LIN {X 0,Y 384.793,Z 555.411,A -85,B 0,C 180,E1 -12841.335,E2 -12841.335} C_VEL
LIN {X 0,Y 382.865,Z 569.469,A -85,B 0,C 180,E1 -12842.535,E2 -12842.535} C_VEL
LIN {X 0,Y 380.828,Z 582.516,A -85,B 0,C 180,E1 -12843.858,E2 -12843.858} C_VEL
LIN {X 0,Y 378.582,Z 595.762,A -85,B 0,C 180,E1 -12845.455,E2 -12845.455} C_VEL
LIN {X 0,Y 376.433,Z 607.881,A -85,B 0,C 180,E1 -12847.207,E2 -12847.207} C_VEL
LIN {X 0,Y 374.348,Z 618.992,A -85,B 0,C 180,E1 -12849.102,E2 -12849.102} C_VEL
LIN {X 0,Y 372.518,Z 629.731,A -85,B 0,C 180,E1 -12851.293,E2 -12851.293} C_VEL
